// TwinCAT 3 PLC project PLC_Skid
// ProgramVersion: 3.1.4026.20
// libraries:
//   Tc2_ControllerToolbox, * (Beckhoff Automation GmbH)
//   Tc2_SerialCom, * (Beckhoff Automation GmbH)
//   Tc2_Standard, * (Beckhoff Automation GmbH)
//   Tc2_System, * (Beckhoff Automation GmbH)
// project tree:
//   / CyclicTaskController.TcTTO, PlcTask.TcTTO, SerialTask.TcTTO
//   DUTs/ EN_AtlasPumpAction.TcDUT, ST_AtlasPumpCmd.TcDUT, ST_AtlasPumpStatus.TcDUT, ST_MassFlowSensor.TcDUT, ST_PressureSensor.TcDUT, ST_Pumps.TcDUT, ST_Valves.TcDUT
//   GVLs/ GVL.TcGVL, GVL_Params.TcGVL, GVL_Serial.TcGVL, IO.TcGVL
//   POUs/General FBs/ FB_MovingAverage.TcPOU, FB_FirstOrderLP.TcPOU, FB_FlowPathCheck.TcPOU, FB_MassFlowMonitor.TcPOU, FB_PressureMonitor.TcPOU, FB_PulseValve.TcPOU, FB_ScaleAnalog.TcPOU, FB_ValvePOS.TcPOU, FB_PumpCTRL.TcPOU, FB_valveCTRL.TcPOU
//   POUs/ MAIN.TcPOU, SerialComm.TcPOU
//   POUs/PID/ PRG_CONTROLLER_CALL.TcPOU, PRG_FB_CTRL_PI.TcPOU
//   POUs/Status FBs/ FB_CheckValveInputs.TcPOU
//   POUs/UnitOp FBs/ FBUO_OPPUMP_AcetonePrime.TcPOU, FBUO_OPFlowFormation.TcPOU, FBUO_OPPump_SyringeSetup.TcPOU, FBUO_OverPressure.TcPOU, FBUO_OverPressure_EX.TcPOU
// real-time tasks:
//   TASK PlcTask: cycle T#10ms, priority 20, ADS port 350
//   TASK CyclicTaskController: cycle T#10ms, priority 1, ADS port 351
//   TASK SerialTask: cycle T#2ms, priority 2, ADS port 352
// I/O:
//   DEVICE Device 1 (EtherCAT), AmsNetId 192.168.43.43.2.1
//     Term 4 (EK1200) [EK1200-5000 EtherCAT Power supply (2A E-Bus)]
//       Term 20 (ELM3104-0020) [ELM3104-0020 4Ch. Ana. Input +/-20mA, 24 bit, high precision, calibrated]
//       Term 22 (EK1122) [EK1122 2 port EtherCAT junction]
//         Term 23 (EK1100) [EK1100 EtherCAT Coupler (2A E-Bus)]
//           Term 24 (EL1409) [EL1409 16Ch. Dig. Input 24V, 3ms]
//           Term 25 (EL2409) [EL2409 16Ch. Dig. Output 24V, 0.5A]
//           Term 26 (EL3078) [EL3078 8Ch. Ana. Input +/-10V, +/-20mA]
//           Term 27 (EL4078) [EL4078 8Ch. Ana. Output, +/-10V, +/-20mA, 16 Bit]
//           Term 12 (EL9011) [EL9011 End Terminal]
//   DEVICE Device 2 (EtherCAT), AmsNetId 192.168.43.43.3.1
//     Term 4 (IOLITE GATE LATCH v2.00 Bus2) [IOLITE GATE LATCH v2.00 Bus2]
//       Term 5 (IOLITEr 6xSTG Bus2) [IOLITEr 6xSTG Bus2]
//       Term 6 (IOLITEr 6xSTG Bus2) [IOLITEr 6xSTG Bus2]
//       Term 7 (IOLITEr 4xCNT Bus2) [IOLITEr 4xCNT Bus2]
//       Term 8 (IOLITEir 8xRTD-HS Bus2) [IOLITEir 8xRTD-HS Bus2]
//       Term 9 (IOLITEr 32xDI Bus2) [IOLITEr 32xDI Bus2]
//       Term 10 (IOLITEr 16xLV Bus2) [IOLITEr 16xLV Bus2]
//       Term 11 (IOLITEr 16xAO Bus2) [IOLITEr 16xAO Bus2]
//       Term 12 (IOLITEr 32xDO Bus2) [IOLITEr 32xDO Bus2]
//       Term 14 (EL9011) [EL9011 End Terminal]
//     Term 13 (IOLITE GATE LATCH v2.00 Bus2) [IOLITE GATE LATCH v2.00 Bus2]
//       Term 14 (IOLITEr 32xDI Bus2) [IOLITEr 32xDI Bus2]
//       Term 15 (IOLITEr 16xLV Bus2) [IOLITEr 16xLV Bus2]
//       Term 16 (IOLITEr 16xAO Bus2) [IOLITEr 16xAO Bus2]
//       Term 15 (EL9011) [EL9011 End Terminal]
// variable links:
//   (this object) <-> Device 1 (EtherCAT)/Term 4 (EK1200)/Term 20 (ELM3104-0020)
//     PlcTask Inputs/IO.AI_wfiFlowMeter <-> PAI Samples 1 Channel 1/Samples[0]
//   (this object) <-> Device 1 (EtherCAT)/Term 4 (EK1200)/Term 22 (EK1122)/Term 23 (EK1100)/Term 24 (EL1409)
//     PlcTask Inputs/IO.DI1_TestManifold <-> DIP Inputs/Input Channel 1
//     PlcTask Inputs/IO.DI2_TestManifold <-> DIP Inputs/Input Channel 2
//   (this object) <-> Device 1 (EtherCAT)/Term 4 (EK1200)/Term 22 (EK1122)/Term 23 (EK1100)/Term 26 (EL3078)
//     PlcTask Inputs/IO.AI1_TestManifold <-> AI Standard (Real32) Channel 1/Value (Real32)
//   (this object) <-> Device 1 (EtherCAT)/Term 4 (EK1200)/Term 22 (EK1122)/Term 23 (EK1100)/Term 27 (EL4078)
//     PlcTask Outputs/IO.AO1_TestManifold <-> AO Standard (Real32) Channel 1/Value (Real32)
//   (this object) <-> Device 2 (EtherCAT)/Term 13 (IOLITE GATE LATCH v2.00 Bus2)/Term 14 (IOLITEr 32xDI Bus2)
//     PlcTask Inputs/IO.DI1_FormManifold <-> AI TxPDO-Map/DI21
//     PlcTask Inputs/IO.DI2_FormManifold <-> AI TxPDO-Map/DI22
//     PlcTask Inputs/IO.DI1_SuspManifold <-> AI TxPDO-Map/DI17
//     PlcTask Inputs/IO.DI2_SuspManifold <-> AI TxPDO-Map/DI18
//     PlcTask Inputs/IO.DI1_dilutionDiV <-> AI TxPDO-Map/DI13
//     PlcTask Inputs/IO.DI2_dilutionDiV <-> AI TxPDO-Map/DI14
//     PlcTask Inputs/IO.DI1_dilutionSV <-> AI TxPDO-Map/DI1
//     PlcTask Inputs/IO.DI2_dilutionSV <-> AI TxPDO-Map/DI2
//     PlcTask Inputs/IO.DI1_formDrain <-> AI TxPDO-Map/DI9
//     PlcTask Inputs/IO.DI2_formDrain <-> AI TxPDO-Map/DI10
//     PlcTask Inputs/IO.DI1_wfiBypassIn <-> AI TxPDO-Map/DI11
//     PlcTask Inputs/IO.DI2_wfiBypassIn <-> AI TxPDO-Map/DI12
//     PlcTask Inputs/IO.DI1_wfiBypassOut <-> AI TxPDO-Map/DI19
//     PlcTask Inputs/IO.DI2_wfiBypassOut <-> AI TxPDO-Map/DI20
//     PlcTask Inputs/IO.DI1_wfiFilterIn <-> AI TxPDO-Map/DI15
//     PlcTask Inputs/IO.DI2_wfiFilterIn <-> AI TxPDO-Map/DI16
//     PlcTask Inputs/IO.DI1_wfiFilterOut <-> AI TxPDO-Map/DI23
//     PlcTask Inputs/IO.DI2_wfiFilterOut <-> AI TxPDO-Map/DI24
//     PlcTask Inputs/IO.DI1_wfiSV <-> AI TxPDO-Map/DI3
//     PlcTask Inputs/IO.DI2_wfiSV <-> AI TxPDO-Map/DI4
//   (this object) <-> Device 2 (EtherCAT)/Term 13 (IOLITE GATE LATCH v2.00 Bus2)/Term 15 (IOLITEr 16xLV Bus2)
//     PlcTask Inputs/IO.AI1_FormManifold <-> UnBuf TxPDO-Map/u9
//     PlcTask Inputs/IO.AI1_SuspManifold <-> UnBuf TxPDO-Map/u11
//     PlcTask Inputs/IO.AI1_dilutionDiV <-> UnBuf TxPDO-Map/u12
//     PlcTask Inputs/IO.AI1_dilutionSV <-> UnBuf TxPDO-Map/u1
//     PlcTask Inputs/IO.AI1_formDrain <-> UnBuf TxPDO-Map/u8
//     PlcTask Inputs/IO.AI1_wfiBypassIn <-> UnBuf TxPDO-Map/u7
//     PlcTask Inputs/IO.AI1_wfiBypassOut <-> UnBuf TxPDO-Map/u10
//     PlcTask Inputs/IO.AI1_wfiFilterIn <-> UnBuf TxPDO-Map/u5
//     PlcTask Inputs/IO.AI1_wfiFilterOut <-> UnBuf TxPDO-Map/u6
//     PlcTask Inputs/IO.AI1_wfiSV <-> UnBuf TxPDO-Map/u2
//   (this object) <-> Device 2 (EtherCAT)/Term 13 (IOLITE GATE LATCH v2.00 Bus2)/Term 16 (IOLITEr 16xAO Bus2)
//     CyclicTaskController Outputs/IO.AO_wfiPump <-> AO RxPDO-Map/AO 3
//     PlcTask Outputs/IO.AO1_FormManifold <-> AO RxPDO-Map/AO 9
//     PlcTask Outputs/IO.AO1_SuspManifold <-> AO RxPDO-Map/AO 11
//     PlcTask Outputs/IO.AO1_dilutionDiV <-> AO RxPDO-Map/AO 12
//     PlcTask Outputs/IO.AO1_dilutionSV <-> AO RxPDO-Map/AO 1
//     PlcTask Outputs/IO.AO1_formDrain <-> AO RxPDO-Map/AO 8
//     PlcTask Outputs/IO.AO1_wfiBypassIn <-> AO RxPDO-Map/AO 7
//     PlcTask Outputs/IO.AO1_wfiBypassOut <-> AO RxPDO-Map/AO 10
//     PlcTask Outputs/IO.AO1_wfiFilterIn <-> AO RxPDO-Map/AO 5
//     PlcTask Outputs/IO.AO1_wfiFilterOut <-> AO RxPDO-Map/AO 6
//     PlcTask Outputs/IO.AO1_wfiSV <-> AO RxPDO-Map/AO 2
//   (this object) <-> Device 2 (EtherCAT)/Term 4 (IOLITE GATE LATCH v2.00 Bus2)/Term 12 (IOLITEr 32xDO Bus2)
//     CyclicTaskController Outputs/IO.DO_wfiPump <-> DO RxPDO-Map/LED 3
//   (this object) <-> Device 2 (EtherCAT)/Term 4 (IOLITE GATE LATCH v2.00 Bus2)/Term 6 (IOLITEr 6xSTG Bus2)
//     PlcTask Inputs/IO.AI_wfiPressureSensor <-> UnBuf TxPDO-Map/u1

CONFIGURATION PLC_Skid
    RESOURCE PLC ON TwinCAT3
        TASK CyclicTaskController(INTERVAL := T#10ms, PRIORITY := 1);
        TASK PlcTask(INTERVAL := T#10ms, PRIORITY := 20);
        TASK SerialTask(INTERVAL := T#2ms, PRIORITY := 2);
        PROGRAM PRG_CONTROLLER_CALL WITH CyclicTaskController : PRG_CONTROLLER_CALL;
        PROGRAM MAIN WITH PlcTask : MAIN;
        PROGRAM SerialComm WITH SerialTask : SerialComm;
    END_RESOURCE
END_CONFIGURATION

// ---- DUTs/EN_AtlasPumpAction.TcDUT
{attribute 'qualified_only'}
{attribute 'strict'}
{attribute 'to_string'}
TYPE EN_AtlasPumpAction :
(
    IDLE := 0,
    STOP_LEFT,
	STOP_RIGHT,
    PAUSE_LEFT,
    PAUSE_RIGHT,
	UNPAUSE_LEFT,
	UNPAUSE_RIGHT,
    EMPTY_LEFT_FAST,
    EMPTY_RIGHT_FAST,
    FILL_LEFT_FAST,
    FILL_RIGHT_FAST,
	EMPTY_LEFT_PRIME,
    EMPTY_RIGHT_PRIME,
    FILL_LEFT_PRIME,
    FILL_RIGHT_PRIME,
	CONTINUOUS
);
END_TYPE

// ---- DUTs/ST_AtlasPumpCmd.TcDUT
TYPE ST_AtlasPumpCmd :
STRUCT
(* Basic Controls *)
    StopLeft        : STRING := 'X0';
	StopRight        : STRING := 'X1';
    PauseLeft       : STRING := 'W0';
	PauseRight       : STRING := 'W1';
    UnpauseLeft     : STRING := 'U0';
	UnpauseRight     : STRING := 'U1';
    (* 15ml/min Port 2 Commands *)
    (* Format: [Command][Volume/Rate] [Port] *)
    EmptyLeft_FAST   	: STRING := 'E0 70000 2';
    EmptyRight_FAST  	: STRING := 'E1 70000 2';
    FillLeft_FAST    	: STRING := 'F0 70000 1';
    FillRight_FAST		: STRING := 'F1 70000 1';
	EmptyLeft_PRIME   	: STRING := 'E0 40000 2';
    EmptyRight_PRIME  	: STRING := 'E1 40000 2';
    FillLeft_PRIME    	: STRING := 'F0 40000 1';
    FillRight_PRIME   	: STRING := 'F1 40000 1';
	CONTINUOUS		  	: STRING := 'C 35000 2 1 0 0';
END_STRUCT
END_TYPE

// ---- DUTs/ST_AtlasPumpStatus.TcDUT
TYPE ST_AtlasPumpStatus :
STRUCT
    (* Parsed from Status Response: #Sn <error> <state> <vol_remain> <movements> <cumul_vol> <flow_rate> <node1> <node2> <total_cumul> *)

    ErrorCode        : INT;         // 0=OK, 1=busy, 2=invalid pump, 3=failure, 4=invalid port, 5=invalid command
    CurrentState     : INT;         // 1=PUMPS_BUSY, 6=PUMPS_IDLE
    VolumeRemaining  : LREAL;       // ul - raw volume remaining from pump (has offset)
    VolumeRemainingCorrected : LREAL; // ul - corrected volume remaining (0 = empty, SyringeSize = full)
    SyringeMovements : DINT;        // Number of syringe movements
    CumulativeVolume : LREAL;       // ul - cumulative volume pumped (may reset)
    CurrentFlowRate  : LREAL;       // ul/min
    NodeSensor1      : STRING(20);  // Node sensor value 1 (or '?' if no node)
    NodeSensor2      : STRING(20);  // Node sensor value 2 (or '?' if no node)
    TotalCumulativeVol : LREAL;     // ul - total cumulative volume (firmware 1.4.26+, persists)

    (* Status Flags *)
    Valid            : BOOL;        // TRUE if last parse succeeded
    IsBusy           : BOOL;        // TRUE if CurrentState = 1 (PUMPS_BUSY)
    IsIdle           : BOOL;        // TRUE if CurrentState = 6 (PUMPS_IDLE)
    HasError         : BOOL;        // TRUE if ErrorCode <> 0

END_STRUCT
END_TYPE

// ---- DUTs/ST_MassFlowSensor.TcDUT
TYPE ST_MassFlowSensor :
STRUCT
	Name : STRING[20];			// Sensor name
	ID : INT;					// Sensor index
	RawValue : REAL;			// Raw input converted from DINT to REAL
	ScaledValue : REAL;			// Scaled engineering units (computed by FB)
	InputMin : REAL;			// Raw input minimum (e.g., 0.0)
	InputMax : REAL;			// Raw input maximum (e.g., 8388607.0 for 24-bit)
	OutputMin : REAL;			// Scaled output minimum (e.g., 0.0)
	OutputMax : REAL;			// Scaled output maximum (e.g., 4500.0 g/min)
	RangeError : BOOL;			// TRUE if raw input outside expected range
	Status : INT;				// 0=OK, 1=Fault
END_STRUCT
END_TYPE

// ---- DUTs/ST_PressureSensor.TcDUT
TYPE ST_PressureSensor :
STRUCT
	Name : STRING[20];			// Sensor name
	ID : INT;					// Sensor index
	RawValue : REAL;			// Raw 4-20mA input from IO
	ScaledValue : REAL;			// Scaled engineering units, unfiltered (computed by FB)
	FilteredValue : REAL;		// Filtered scaled value (used for control/protection)
	FilterTimeConst : REAL;		// Low-pass filter time constant in seconds (0.0 = no filtering)
	InputMin : REAL;			// Raw input minimum (e.g., 4.0)
	InputMax : REAL;			// Raw input maximum (e.g., 20.0)
	OutputMin : REAL;			// Scaled output minimum (e.g., 0.0)
	OutputMax : REAL;			// Scaled output maximum (e.g., 30.0)
	RangeError : BOOL;			// TRUE if raw input outside expected range
	Status : INT;				// 0=OK, 1=Fault
END_STRUCT
END_TYPE

// ---- DUTs/ST_Pumps.TcDUT
TYPE ST_Pumps :
STRUCT
	Name : STRING[20]; 		// Pump Name
	ID : INT;					// Pump index
	IsOn : BOOL;				// Command: TRUE = pump active
	CMDVoltage : REAL;			// Command: speed setpoint 0-10V
	ControllerIsOn : BOOL;			// Allows for PID Control
	ControllerSetppoint : REAL;		//Setpoint mass flow rate in g/min
	DO1 : BOOL := FALSE;				// Output: digital on/off (computed by FB_PumpCTRL)
	AO1 : REAL := 0;				// Output: analog voltage (computed by FB_PumpCTRL)
	PressureValue : REAL;			// Current pressure reading (mapped from sensor in MAIN)
	PressureLimit : REAL;			// Overpressure trip threshold (0.0 = no check)
	OverPressure : BOOL;			// Latching overpressure flag (clear from HMI to reset)
	FlowPathOpen : BOOL;			// TRUE if required flow path valves are confirmed open
	Status : INT;				// 0=OK, 1=Fault
END_STRUCT
END_TYPE

// ---- DUTs/ST_Valves.TcDUT
TYPE ST_Valves :
STRUCT
    Name : WSTRING(80); // Descriptive name (e.g., 'ValveA', 'InletValve1')
	ID : INT;	// Valve Index
    DI1 : BOOL; // Valve open feedback (if True Valve Open)
    DI2 : BOOL; // Valve closed feedback (if True Valve Close)
    DO1 : BOOL; // Valve Initialization Signal
    AI1 : REAL; // Valve position (0-10V)
    AO1 : REAL; // Valve setpoint (0-10V)
    State : INT; // Operating state (0=Off, 1=Open/Close, 2=OpenLoop, 3=PID)
    isOpen : BOOL; // HMI open/close input
    Setpoint : REAL; // Setpoint for OpenLoop or PID (0-10V)
    PV : REAL; // Process Variable for PID
    Output : REAL; // PID output (0-10V)
	Status : INT; // Diagnostic status (0 = OK, 1 = Fault)
END_STRUCT
END_TYPE

// ---- GVLs/GVL.TcGVL
VAR_GLOBAL CONSTANT
	valveCount : INT := 11;
	sValveNames : ARRAY[1..valveCount] OF WSTRING := 	["Dilution Selector", 
														"WFI Selector", 
														"Formation Drain", 
														"WFI Filter Bypass Inlet",
														"WFI Filter Inlet",
														"WFI Filter Outlet",
														"WFI Filter Bypass Outlet",
														"Dilution Diverter",
														"Formation Manifold",
														"Suspension Manifold",
														"Test Manifold"];													
stValveID : ARRAY[1..valveCount] OF INT := 	[1, 	// Dilution Selector
											 2, 		// WFI Selector,
											 3, 		// Formation Drain,
											 4, 		// WFI Filter Bypass Inlet,
											 5, 		// WFI Filter Inlet,
											 6, 		// WFI Filter Outlet,
											 7, 		// WFI Filter Bypass Outlet,
											 8, 		// Dilution Diverter,
											 9, 		// Formation Manifold,
											 10, 	// Suspension Manifold,
											 11		// Test Manifold
											];
											
pumpCount : INT := 2;
sPumpNames : ARRAY[1..pumpCount] OF WSTRING := 		
	["WFI Pump", "Suspension Pump"];

pressureSensorCount : INT := 3;
sPressureSensorNames : ARRAY[1..pressureSensorCount] OF WSTRING :=
	["WFI Pressure", "Suspension Pressure", "TFF Outlet Pressure"];

massFlowSensorCount : INT := 3;
sMassFlowSensorNames : ARRAY[1..massFlowSensorCount] OF WSTRING :=
	["WFI Mass Flow", "Suspension Mass Flow", "Discharge Flow"];
	
	
END_VAR

VAR_GLOBAL

	myText 		: STRING(16) := 'Type';
	myNum		: REAL := 0;
	avg10WFI_MassFlowRate : REAL;
	
	fSetpointValueToScope			: LREAL;
	fActualValueToScope				: LREAL;
	fOutToScope						: LREAL;
	
END_VAR

// ---- GVLs/GVL_Params.TcGVL
{attribute 'qualified_only'}
VAR_GLOBAL
	


END_VAR

// ---- GVLs/GVL_Serial.TcGVL
{attribute 'qualified_only'}
VAR_GLOBAL
    (* I/O variables for a PC-COM port *)
    stIn_PcCom      AT %I*  : PcComInData;  (* linked to the port in the TwinCAT System Manager *)
    stOut_PcCom     AT %Q*  : PcComOutData; (* linked to the port in the TwinCAT System Manager *)
    RxBufferPcCom           : ComBuffer;    (* Receive data buffer *)
    TxBufferPcCom           : ComBuffer;    (* Transmit data buffer *)

    (* PC Control *)
    bEnablePCControl    : BOOL := FALSE;    // Set TRUE to enable PC Control mode
    sCommandString      : STRING := '';     // Manual command string (set before bStartCommand)
    bStartCommand       : BOOL;             // Trigger to send manual command via sCommandString
    eSelectedAction     : EN_AtlasPumpAction := EN_AtlasPumpAction.IDLE;

    (* Pump Status - Updated every 50ms per axis (100ms total cycle) *)
    stPumpStatus        : ARRAY[0..1] OF ST_AtlasPumpStatus;  // Status for axis 0 and axis 1
    bStatusPollingActive: BOOL := FALSE;    // TRUE when status polling is running

    (* Syringe Configuration - used to correct VolumeRemaining offset *)
    (* Each axis may have a different "full" reference point from the pump *)
    (* Axis 0: Full=5000, Empty=-20000  -> Offset = 20000 (or SyringeSize - FullRef) *)
    (* Axis 1: Full=10000, Empty=-15000 -> Offset = 15000 (or SyringeSize - FullRef) *)
    (* Corrected = Raw + Offset, so that Full=SyringeSize, Empty=0 *)
    rSyringeSize        : ARRAY[0..1] OF LREAL := [25000.0, 25000.0];  // ul - syringe size for each axis
    rFullReference      : ARRAY[0..1] OF LREAL := [5000.0, 10000.0];   // ul - raw value when syringe is full

END_VAR

// ---- GVLs/IO.TcGVL
{attribute 'qualified_only'}
VAR_GLOBAL
	

//----------------------------------DO Place Holder INIT valve 1 -------------------------------------------------//
	//AO1 AT %Q* : REAL;
	DO1 AT %Q* : BOOL;
//---------------------------------------------------------------------------------------------------------------//
	
//---------------------------------- PUMP MAPPING -------------------------------------------------//
	// WFI Pump (index 1)
	DO_wfiPump AT %Q* : BOOL;			// Digital Output for turning pump on and off
	AO_wfiPump AT %Q* : REAL;			// Analog Output for pump speed control
	// Suspension Pump (index 2) - not yet connected
	// DO_suspPump AT %Q* : BOOL;		// Digital Output for turning pump on and off
	// AO_suspPump AT %Q* : REAL;		// Analog Output for pump speed control
//-------------------------------------------------------------------------------------------------//

//---------------------------------- PRESSURE SENSOR MAPPING ----------------------------------------//
	// WFI Pressure Sensor (index 1)
	AI_wfiPressureSensor AT %I* : REAL;			// Analog Input for WFI pressure sensor (4-20mA)
	// Suspension Pressure Sensor (index 2) - not yet connected
	// AI_suspPressureSensor AT %I* : REAL;
	// TFF Outlet Pressure Sensor (index 3) - not yet connected
	// AI_tffOutletPressureSensor AT %I* : REAL;
//-------------------------------------------------------------------------------------------------//

//---------------------------------- MASS FLOW METER MAPPING ------------------------------------------//
	// WFI Mass Flow Meter (index 1)
	AI_wfiFlowMeter AT %I* : DINT;				// Coriolis meter raw input (24-bit DINT)
	// Suspension Mass Flow Meter (index 2) - not yet connected
	// AI_suspMassFlowMeter AT %I* : DINT;
	// Discharge Flow Meter (index 3) - not yet connected
	// AI_dischargeFlowMeter AT %I* : DINT;
//-------------------------------------------------------------------------------------------------//

//---------------------------------- VALVE MAPPING ------------------------------------------------//
	// IOs Dilution Selector Valve (SV)
    DI1_dilutionSV AT %I* : BOOL; 		// Digital Input 1 Closed Feedback
    DI2_dilutionSV AT %I* : BOOL; 		// Digital Input 2 Open Feedback
    AI1_dilutionSV AT %I* : REAL;  		// Analog Input 1 Valve Position Feedback
    DO1_dilutionSV AT %Q* : BOOL; 		// Digital Output 1 Valve Initialization
    AO1_dilutionSV AT %Q* : REAL; 		// Analog Output 1 Valve Position Control Variable (0-10V)
    
    // IOs WFI Selector Valve (SV) 
    DI1_wfiSV AT %I* : BOOL;      		// Digital Input 1 Closed Feedback
    DI2_wfiSV AT %I* : BOOL;      		// Digital Input 2 Open Feedback
    AI1_wfiSV AT %I* : REAL;       		// Analog Input 1 Valve Position Feedback
    DO1_wfiSV AT %Q* : BOOL;     		// Digital Output 1 Valve Initialization
    AO1_wfiSV AT %Q* : REAL;      		// Analog Output 1 Valve Position Control Variable (0-10V)

	// IOs Formation Drain Valve 
    DI1_formDrain AT %I* : BOOL;      	// Digital Input 1 Closed Feedback
    DI2_formDrain AT %I* : BOOL;      	// Digital Input 2 Open Feedback
    AI1_formDrain AT %I* : REAL;       	// Analog Input 1 Valve Position Feedback
    DO1_formDrain AT %Q* : BOOL;     	// Digital Output 1 Valve Initialization
    AO1_formDrain AT %Q* : REAL;      	// Analog Output 1 Valve Position Control Variable (0-10V)
	
	// IOs WFI Bypass Inlet Valve
    DI1_wfiBypassIn AT %I* : BOOL;      // Digital Input 1 Closed Feedback
    DI2_wfiBypassIn AT %I* : BOOL;      // Digital Input 2 Open Feedback
    AI1_wfiBypassIn AT %I* : REAL;      // Analog Input 1 Valve Position Feedback
    DO1_wfiBypassIn AT %Q* : BOOL;     	// Digital Output 1 Valve Initialization
    AO1_wfiBypassIn AT %Q* : REAL;      // Analog Output 1 Valve Position Control Variable (0-10V)
	
		// IOs WFI Filter Inlet Valve
    DI1_wfiFilterIn AT %I* : BOOL;      // Digital Input 1 Closed Feedback
    DI2_wfiFilterIn AT %I* : BOOL;      // Digital Input 2 Open Feedback
    AI1_wfiFilterIn AT %I* : REAL;      // Analog Input 1 Valve Position Feedback
    DO1_wfiFilterIn AT %Q* : BOOL;     	// Digital Output 1 Valve Initialization
    AO1_wfiFilterIn AT %Q* : REAL;      // Analog Output 1 Valve Position Control Variable (0-10V)
	
		// IOs WFI Filter Outlet Valve
    DI1_wfiFilterOut AT %I* : BOOL;      // Digital Input 1 Closed Feedback
    DI2_wfiFilterOut AT %I* : BOOL;      // Digital Input 2 Open Feedback
    AI1_wfiFilterOut AT %I* : REAL;      // Analog Input 1 Valve Position Feedback
    DO1_wfiFilterOut AT %Q* : BOOL;     	// Digital Output 1 Valve Initialization
    AO1_wfiFilterOut AT %Q* : REAL;      // Analog Output 1 Valve Position Control Variable (0-10V)
	
		// IOs WFI Bypass Outlet Valve
    DI1_wfiBypassOut AT %I* : BOOL;      // Digital Input 1 Closed Feedback
    DI2_wfiBypassOut AT %I* : BOOL;      // Digital Input 2 Open Feedback
    AI1_wfiBypassOut AT %I* : REAL;      // Analog Input 1 Valve Position Feedback
    DO1_wfiBypassOut AT %Q* : BOOL;     	// Digital Output 1 Valve Initialization
    AO1_wfiBypassOut AT %Q* : REAL;      // Analog Output 1 Valve Position Control Variable (0-10V)
	
		// IOs Dilution Diverter Valve
    DI1_dilutionDiV AT %I* : BOOL;      // Digital Input 1 Closed Feedback
    DI2_dilutionDiV AT %I* : BOOL;      // Digital Input 2 Open Feedback
    AI1_dilutionDiV AT %I* : REAL;      // Analog Input 1 Valve Position Feedback
    DO1_dilutionDiV AT %Q* : BOOL;     	// Digital Output 1 Valve Initialization
    AO1_dilutionDiV AT %Q* : REAL;      // Analog Output 1 Valve Position Control Variable (0-10V)
	
		// IOs Formation Manifold Valve
    DI1_FormManifold AT %I* : BOOL;      // Digital Input 1 Closed Feedback
    DI2_FormManifold AT %I* : BOOL;      // Digital Input 2 Open Feedback
    AI1_FormManifold AT %I* : REAL;      // Analog Input 1 Valve Position Feedback
    DO1_FormManifold AT %Q* : BOOL;     	// Digital Output 1 Valve Initialization
    AO1_FormManifold AT %Q* : REAL;      // Analog Output 1 Valve Position Control Variable (0-10V)
	
		// IOs Suspension Manifold Valve
    DI1_SuspManifold AT %I* : BOOL;      // Digital Input 1 Closed Feedback
    DI2_SuspManifold AT %I* : BOOL;      // Digital Input 2 Open Feedback
    AI1_SuspManifold AT %I* : REAL;      // Analog Input 1 Valve Position Feedback
    DO1_SuspManifold AT %Q* : BOOL;     	// Digital Output 1 Valve Initialization
    AO1_SuspManifold AT %Q* : REAL;      // Analog Output 1 Valve Position Control Variable (0-10V)
	
			// IOs Test Manifold Valve
    DI1_TestManifold AT %I* : BOOL;      // Digital Input 1 Closed Feedback
    DI2_TestManifold AT %I* : BOOL;      // Digital Input 2 Open Feedback
    AI1_TestManifold AT %I* : REAL;      // Analog Input 1 Valve Position Feedback (4-20ma)
    DO1_TestManifold AT %Q* : BOOL;     	// Digital Output 1 Valve Initialization
    AO1_TestManifold AT %Q* : REAL;      // Analog Output 1 Valve Position Control Variable (4-20ma)
//-------------------------------------------------------------------------------------------------//

END_VAR

// ---- POUs/PID/PRG_CONTROLLER_CALL.TcPOU
PROGRAM PRG_CONTROLLER_CALL

VAR
	
	stPumps 	: ARRAY[1..GVL.pumpCount] OF ST_Pumps;
	
	
END_VAR




IF stPumps[1].ControllerIsOn AND stPumps[1].IsOn THEN
	IO.DO_wfiPump 					:= TRUE;
	PRG_FB_CTRL_PI();

	ELSE
	IO.DO_wfiPump := FALSE;
	IO.AO_wfiPump := stPumps[1].ControllerSetppoint := 0;
END_IF

END_PROGRAM

// ---- POUs/PID/PRG_FB_CTRL_PI.TcPOU
PROGRAM PRG_FB_CTRL_PI


VAR
	stPumps 	: ARRAY[1..GVL.pumpCount] OF ST_Pumps;	

	fSetpointValue				: LREAL;
	fActualValue				: LREAL;
	fManSyncValue				: LREAL;
	bSync						: BOOL;

	fOut						: LREAL;
	bHold						: BOOL;

	eMode						: E_CTRL_MODE;
	stCTRL_PI_PARAMS			: ST_CTRL_PI_PARAMS;

	eErrorId					: E_CTRL_ERRORCODES;
	bError						: BOOL;
	bARWactive					: BOOL;

	(* controller  *)
	fbCTRL_PI					: FB_CTRL_PI;

	bInit						: BOOL := TRUE;
	fbTON						: TON;
END_VAR

IF bInit THEN
	(* init parameter struct *)
	stCTRL_PI_PARAMS.tCtrlCycleTime		:= T#10MS;
	stCTRL_PI_PARAMS.tTaskCycleTime		:= T#10MS;
	stCTRL_PI_PARAMS.tTn				:= T#2S;	(* derivative gain Tv				*)
	stCTRL_PI_PARAMS.fKp				:= 2;		(* proportional gain Kp				*)
	stCTRL_PI_PARAMS.fOutMaxLimit		:= 3;  		(* maximum output limit				*)
	stCTRL_PI_PARAMS.fOutMinLimit		:= 0;		(* minimum output limit				*)

	(* set the mode to ACTIVE --> normal operation *)
	eMode := eCTRL_MODE_ACTIVE;

	(* reset the init flag *)
	bInit := FALSE;
END_IF

fSetpointValue := stPumps[1].ControllerSetppoint;
fActualValue := GVL.avg10WFI_MassFlowRate;

(* copy var to scope var *)
fSetpointValueToScope 		:= fSetpointValue;
fActualValueToScope 		:= fActualValue;

(* call controller *)
fbCTRL_PI(		fSetpointValue		:= fSetpointValue,
					fActualValue		:= fActualValue,
					fManSyncValue	:= fManSyncValue,
					bSync				:= bSync,
					eMode				:= eMode,
					bHold				:= bHold,
					stParams			:= stCTRL_PI_PARAMS,
					fOut				=> fOut,
					bARWactive		=> bARWactive,
					eErrorId			=> eErrorId,
					bError				=> bError
				);


(* copy var to scope var *)
fOut := stPumps[1].CMDVoltage;
fOutToScope := fOut;

END_PROGRAM

// ---- POUs/MAIN.TcPOU
PROGRAM MAIN
VAR
//-------------------- Program Initialization Variables ----------------------------//
	i : INT; //Initialization Counter
	CycleCount : INT := 0; // Cycle counter
	Initialized : BOOL := FALSE; // Flag for initialization
	CtrlStatus : INT; // Status output
//----------------------------------------------------------------------------------//


//--------------------------------- Struct Init ------------------------------------//
// Constant array of valve names
	stValves : ARRAY[1..GVL.valveCount] OF ST_Valves;
	stPumps : ARRAY[1..GVL.pumpCount] OF ST_Pumps;
	stPressureSensors : ARRAY[1..GVL.pressureSensorCount] OF ST_PressureSensor;
	stMassFlowSensors : ARRAY[1..GVL.massFlowSensorCount] OF ST_MassFlowSensor;
//----------------------------------------------------------------------------------//


//----------------------------INIT Function Blocks----------------------------------//
	systemCheck_Valves : FB_CheckValveInputs;
	valveCtrl : FB_valveCTRL;
	pumpCtrl : FB_PumpCTRL;
	varPulse : FB_PulseValve;   // Instance of the function block
	unitOp_OverPressure : FBUO_OverPressure;
	unitOp_OverPressureEX : FBUO_OverPressure_EX;
	pressureMonitor : FB_PressureMonitor;
	massFlowMonitor : FB_MassFlowMonitor;
	flowPathCheck_WFI : FB_FlowPathCheck;
	wfi_MassFlowAvg10 : FB_MovingAverage;
	wfi_MassFlowAvg30 : FB_MovingAverage;
	wfi_MassFlowAvg100 : FB_MovingAverage;
//----------------------------------------------------------------------------------//	
	
//---------------------------- General Variables -----------------------------------//
	outputDO1 : BOOL;           // Local output variable
    tPulseTime : TIME := T#1000MS; // Pulse duration
	//avg10WFI_MassFlowRate : REAL;
	avg30WFI_MassFlowRate : REAL;
	avg100WFI_MassFlowRate : REAL;
	
//---------------------INIT Control Variables---------------------------------------//
	hOP_ProcessState			: BOOL	:= TRUE;	// Overpressure process step active
	hOP_ValvesPositionSet	 	: BOOL 	:= TRUE;	// Position Valves
	hOP_PumpActive				: BOOL	:= FALSE;	// Turn on Pump
	hOP_PumpSpeed				: REAL 	:= 0;		// Pump Speed
//----------------------------------------------------------------------------------//

//---------------------INIT Control Variables---------------------------------------//
	hOPEX_ProcessState			: BOOL	:= FALSE;	// Overpressure process step active
	hOPEX_ValvesPositionSet	 	: BOOL 	:= FALSE;	// Position Valves
	hOPEX_PumpActive			: BOOL	:= FALSE;	// Turn on Pump
//----------------------------------------------------------------------------------//

//---------------------Flow Path Definitions---------------------------------------//
	wfiFlowPath_OP		: ARRAY[1..GVL.valveCount] OF INT := [2,5,0,0,0,0,0,0,0,0];
	wfiFlowPath_OPEX	: ARRAY[1..GVL.valveCount] OF INT := [2,4,7,8,9,10,0,0,0,0];
	wfiActiveFlowPath	: ARRAY[1..GVL.valveCount] OF INT;
//----------------------------------------------------------------------------------//


//----------------------------INIT Function Blocks----------------------------------//
	fbSyringeSetup : FBUO_OPPump_SyringeSetup;
	fbAcetonePrime : FBUO_OPPump_AcetonePrime;
	fbFlowFormation : FBUO_OPFlowFormation;
//----------------------------------------------------------------------------------//

///---------------------Organic Phase Setup ---------------------------------------//
OPActive					: BOOL	:= FALSE;
bStartSyringeSetup			: BOOL	:= FALSE;	// Start Syringe Setup Routine
bStartActenePriming			: BOOL	:= FALSE;	// Start Acetone Priming Routine
bStartFlowFormation			: BOOL	:= FALSE;	// Start/Stop Continuous Flow Formation
nAcetoneCycles				: INT	:= 2;
nAcetoneCycle				: INT;	
//----------------------------------------------------------------------------------//

// -----------------------MATLAB Variables for testing ----------------------------//
mtbIN		: INT		:= 1000;
mtbOUT		: INT;
mtbActive	: BOOL		:= FALSE;	
currentValue : REAL := 0;
END_VAR

//------------------------------------Process Code ----------------------------------------//
//---------------------------------- Initialization----------------------------------------//
IF NOT Initialized THEN
    FOR i := 1 TO gvl.valveCount DO
        stValves[i].Name := GVL.sValveNames[i]; // Assign valve names
		stValves[i].ID := GVL.stValveID[i];
        stValves[i].State := 0; // Initialize to Closed
        stValves[i].AO1 := 0.0; // Closed position
        stValves[i].Status := 0; // No faults
        stValves[i].isOpen := FALSE; // Initialize to closed
    END_FOR
	FOR i := 1 TO GVL.pumpCount DO
		stPumps[i].Name := WSTRING_TO_STRING(GVL.sPumpNames[i]);
		stPumps[i].ID := i;
		stPumps[i].IsOn := FALSE;
		stPumps[i].CMDVoltage := 0.0;
		stPumps[i].ControllerIsOn := FALSE;
		stPumps[i].DO1 := FALSE;
		stPumps[i].AO1 := 0.0;
		stPumps[i].PressureValue := 0.0;
		stPumps[i].PressureLimit := 10.0;
		stPumps[i].OverPressure := FALSE;
		stPumps[i].FlowPathOpen := FALSE;
		stPumps[i].Status := 0;
	END_FOR
	FOR i := 1 TO GVL.pressureSensorCount DO
		stPressureSensors[i].Name := WSTRING_TO_STRING(GVL.sPressureSensorNames[i]);
		stPressureSensors[i].ID := i;
		stPressureSensors[i].RawValue := 0.0;
		stPressureSensors[i].ScaledValue := 0.0;
		stPressureSensors[i].FilteredValue := 0.0;
		stPressureSensors[i].FilterTimeConst := 0.1;
		stPressureSensors[i].InputMin := 4.0;
		stPressureSensors[i].InputMax := 20.0;
		stPressureSensors[i].OutputMin := 0.0;
		stPressureSensors[i].OutputMax := 30.0;
		stPressureSensors[i].RangeError := FALSE;
		stPressureSensors[i].Status := 0;
	END_FOR
	FOR i := 1 TO GVL.massFlowSensorCount DO
		stMassFlowSensors[i].Name := WSTRING_TO_STRING(GVL.sMassFlowSensorNames[i]);
		stMassFlowSensors[i].ID := i;
		stMassFlowSensors[i].RawValue := 0.0;
		stMassFlowSensors[i].ScaledValue := 0.0;
		stMassFlowSensors[i].InputMin := 0;
		stMassFlowSensors[i].InputMax := 8388607.0;
		stMassFlowSensors[i].OutputMin := 0.0;
		stMassFlowSensors[i].OutputMax := 4500.0;
		stMassFlowSensors[i].RangeError := FALSE;
		stMassFlowSensors[i].Status := 0;
	END_FOR
    Initialized := TRUE;
END_IF
CycleCount := CycleCount + 1;

//--------------------------------------------------------------------------------------------//


//------------------------------ Valve Position Monitoring -----------------------------------//
systemCheck_Valves(
	fbCheckProcessState := TRUE, 
	fbValves 			:= stValves);
//--------------------------------------------------------------------------------------------//

//------------------------------- Flow Path Check --------------------------------------------//
// Select active flow path based on which operation is running
IF hOP_ProcessState THEN
	wfiActiveFlowPath := wfiFlowPath_OP;
ELSIF hOPEX_ProcessState THEN
	wfiActiveFlowPath := wfiFlowPath_OPEX;
END_IF
// Check if required valves are confirmed open
flowPathCheck_WFI(
	fbRequiredValves := wfiActiveFlowPath,
	fbValves := stValves);
stPumps[1].FlowPathOpen := flowPathCheck_WFI.fbPathOpen;
//------------------------------------------------------------------------------------------//

//------------------------- Overpressure Process (Development Only) --------------------------//
unitOp_OverPressureEX(
	fbOPprocessState 		:= hOPEX_ProcessState,
	fbValvePositionReady 	:= hOPEX_ValvesPositionSet, 
	fbValves 				:= stValves);
//--------------------------------------------------------------------------------------------//


//------------------------- Overpressure Process (Development Only) --------------------------//
unitOp_OverPressure(
	fbOPprocessState 		:= hOP_ProcessState,
	fbValvePositionReady 	:= hOP_ValvesPositionSet, 
	fbValves 				:= stValves,
	fbPumpActive			:=hOP_PumpActive,
	fbPumpSpeed				:= hOP_PumpSpeed);
//--------------------------------------------------------------------------------------------//

//---------------------------------- Atlas Syringe Setup--------------------------------------//
GVL_Serial.bEnablePCControl := OPActive;
IF OPActive THEN
  fbSyringeSetup(
      bEnable := TRUE,
      bStart  := bStartSyringeSetup
  );
//--------------------------------------------------------------------------------------------//  

//---------------------------------- Acetone Priming -----------------------------------------//
  fbAcetonePrime(
      bEnable            := TRUE,
      bStartAcetonePrime := bStartActenePriming,
      nSyringeCycles     := nAcetoneCycles
  );
  // Monitor progress
  nAcetoneCycle := fbAcetonePrime.nCurrentCycle;  // Shows 1, then 2

//---------------------------------- Continuous Flow Formation --------------------------------//
  fbFlowFormation(
      bEnable := TRUE,
      bStart  := bStartFlowFormation
  );
END_IF
//--------------------------------------------------------------------------------------------// 

//OP Routine Status
  IF fbSyringeSetup.bDone THEN
      // Syringes at 12.5ml - ready for operator to attach
  END_IF

  IF fbAcetonePrime.bDone THEN
      // Priming complete, syringes are empty
  END_IF

//------------------------------ Pressure Monitoring ----------------------------------------//
// Pressure Sensor I/O Mapping
stPressureSensors[1].RawValue := IO.AI_wfiPressureSensor;
// stPressureSensors[2].RawValue := IO.AI_suspPressureSensor;       // uncomment when wired
// stPressureSensors[3].RawValue := IO.AI_tffOutletPressureSensor;  // uncomment when wired
pressureMonitor(fbSensors := stPressureSensors);
//---------------------------------------------------------------------------------------------//

//----------------------------- Mass Flow Monitoring -----------------------------------------------------//					
// Mass Flow Sensor I/O Mapping (DINT to REAL conversion at boundary)
stMassFlowSensors[1].RawValue := DINT_TO_REAL(IO.AI_wfiFlowMeter);
// stMassFlowSensors[2].RawValue := DINT_TO_REAL(IO.AI_suspMassFlowMeter);     // uncomment when wired
// stMassFlowSensors[3].RawValue := DINT_TO_REAL(IO.AI_dischargeFlowMeter);    // uncomment when wired
massFlowMonitor(fbSensors := stMassFlowSensors);

// 10-sample moving average for WFI mass flow rate
wfi_MassFlowAvg10(
	fbInputValue := stMassFlowSensors[1].ScaledValue,
	fbSampleSize := 10,
	fbAverageValue => GVL.avg10WFI_MassFlowRate);

// 30-sample moving average for WFI mass flow rate
wfi_MassFlowAvg30(
	fbInputValue := stMassFlowSensors[1].ScaledValue,
	fbSampleSize := 30,
	fbAverageValue => avg30WFI_MassFlowRate);

// 100-sample moving average for WFI mass flow rate
wfi_MassFlowAvg100(
	fbInputValue := stMassFlowSensors[1].ScaledValue,
	fbSampleSize := 100,
	fbAverageValue => avg100WFI_MassFlowRate);
//-----------------------------------------------------------------------------------------------------//

//------------------------------- Pump Control ------------------------------------//
// Map filtered pressure readings to pumps for overpressure protection
stPumps[1].PressureValue := stPressureSensors[1].FilteredValue;	// WFI Pump <- WFI Pressure
stPumps[2].PressureValue := stPressureSensors[2].FilteredValue;	// Suspension Pump <- Suspension Pressure
pumpCtrl(fbPumps := stPumps);
// WFI Pump I/O Mapping (index 1)
IF mtbActive AND NOT stPumps[1].ControllerIsOn THEN
	IO.DO_wfiPump := stPumps[1].DO1;
	IO.AO_wfiPump := stPumps[1].AO1;
	ELSE
	IO.DO_wfiPump := FALSE;
	IO.AO_wfiPump := 0;
END_IF
// Suspension Pump I/O Mapping (index 2) - uncomment when I/O available
// IO.DO_suspPump := stPumps[2].DO1;
// IO.AO_suspPump := stPumps[2].AO1;
//--------------------------------------------------------------------------------------------------------------//

//------------------------------- Matlab Testing ---------------------------------------------------------------//

IF mtbActive AND mtbOut <500 THEN
	mtbOut := mtbOut+mtbIN;
	ELSE
	mtbOut :=0;
END_IF
IO.AO1_TestManifold := currentValue;
//--------------------------------------------------------------------------------------------------------------//

//------------------------------- Valve Init Function (To be refined later) ------------------------------------//
// Correct function block call with inputs
varPulse(Valve := outputDO1, pulseTime := tPulseTime);
// Assign output to global I/O
IO.DO1_dilutionSV := outputDO1;
//-----------------------------------------------------------------------------------------------------//

//-----------------------------Process Code END ----------------------------------------//

END_PROGRAM

// ---- POUs/Status FBs/FB_CheckValveInputs.TcPOU
FUNCTION_BLOCK FB_CheckValveInputs
VAR_INPUT
	fbCheckProcessState :	BOOL;
END_VAR
VAR_IN_OUT
    fbValves : ARRAY[1..GVL.valveCount] OF ST_Valves;
END_VAR
VAR_OUTPUT
	
END_VAR
VAR
	
END_VAR

IF fbCheckProcessState THEN
	fbValves[1].DI1 := IO.DI1_dilutionSV;
	fbValves[1].AI1 := IO.AI1_dilutionSV;
	fbValves[1].DI2 := IO.DI2_dilutionSV;

	fbValves[2].DI1 := IO.DI1_wfiSV;
	fbValves[2].AI1 := IO.AI1_wfiSV;
	fbValves[2].DI2 := IO.DI2_wfiSV;

	fbValves[3].DI1 := IO.DI1_formDrain;
	fbValves[3].AI1 := IO.AI1_formDrain;
	fbValves[3].DI2 := IO.DI2_formDrain;

	fbValves[4].DI1 := IO.DI1_wfiBypassIn;
	fbValves[4].AI1 := IO.AI1_wfiBypassIn;
	fbValves[4].DI2 := IO.DI2_wfiBypassIn;
	
	fbValves[5].DI1 := IO.DI1_wfiFilterIn;
	fbValves[5].AI1 := IO.AI1_wfiFilterIn;
	fbValves[5].DI2 := IO.DI2_wfiFilterIn;
	
	fbValves[6].DI1 := IO.DI1_wfiFilterOut;
	fbValves[6].AI1 := IO.AI1_wfiFilterOut;
	fbValves[6].DI2 := IO.DI2_wfiFilterOut;
	
	fbValves[7].DI1 := IO.DI1_wfiBypassOut;
	fbValves[7].AI1 := IO.AI1_wfiBypassOut;
	fbValves[7].DI2 := IO.DI2_wfiBypassOut;
	
	fbValves[8].DI1 := IO.DI1_dilutionDiV;
	fbValves[8].AI1 := IO.AI1_dilutionDiV;
	fbValves[8].DI2 := IO.DI2_dilutionDiV;
	
	fbValves[9].DI1 := IO.DI1_FormManifold;
	fbValves[9].AI1 := IO.AI1_FormManifold;
	fbValves[9].DI2 := IO.DI2_FormManifold;
	
	fbValves[10].DI1 := IO.DI1_SuspManifold;
	fbValves[10].AI1 := IO.AI1_SuspManifold;
	fbValves[10].DI2 := IO.DI2_SuspManifold;
END_IF

END_FUNCTION_BLOCK

// ---- POUs/General FBs/FB_valveCTRL.TcPOU
FUNCTION_BLOCK FB_valveCTRL
VAR_INPUT
    //fbValveNames : ARRAY[1..GVL.valveCount] OF STRING[20]; // Array of valve names
END_VAR
VAR_IN_OUT
    fbValves : ARRAY[1..GVL.valveCount] OF ST_Valves;   // Array of valve structures
END_VAR
VAR_OUTPUT
    //Status : INT;                             // 0=OK, 1=Valve not found
END_VAR
VAR
    i : INT;                                  // Internal loop variable
END_VAR

// Initialize output
//Status := 0;

// Control valves based on hOpenClose
FOR i := 1 TO gvl.valveCount DO
    //IF fbValves[i].Name = fbValveNames[i] THEN
        CASE fbValves[i].State OF
            1: // Open/Close mode
                IF fbValves[i].isOpen THEN
                    fbValves[i].AO1 := 10.0; // Open
                ELSE
                    fbValves[i].AO1 := 0.0; // Close
                END_IF
            2: // OpenLoop
                fbValves[i].AO1 := fbValves[i].Setpoint;
            3: // PID (Placeholder)
                fbValves[i].AO1 := 0.0;
            ELSE
                fbValves[i].AO1 := 0.0;
                //Status := Status + 2;
        END_CASE
    //ELSE
        //Status := Status + 1;
    //END_IF
END_FOR

END_FUNCTION_BLOCK

// ---- POUs/General FBs/FB_PumpCTRL.TcPOU
FUNCTION_BLOCK FB_PumpCTRL
VAR_INPUT
END_VAR
VAR_IN_OUT
    fbPumps : ARRAY[1..GVL.pumpCount] OF ST_Pumps;   // Array of pump structures
END_VAR
VAR_OUTPUT
END_VAR
VAR
    i : INT;                                  // Internal loop variable
END_VAR

// Pump control - open loop voltage command with overpressure protection
FOR i := 1 TO GVL.pumpCount DO
	// Overpressure latch: trips when pressure >= limit, stays latched until cleared externally
	IF fbPumps[i].PressureLimit > 0.0 AND fbPumps[i].PressureValue >= fbPumps[i].PressureLimit THEN
		fbPumps[i].OverPressure := TRUE;
	END_IF

	// Control pump output (safety checks: overpressure, flow path)
	IF fbPumps[i].OverPressure THEN
		fbPumps[i].DO1 := FALSE;
		fbPumps[i].AO1 := 0.0;
	ELSIF NOT fbPumps[i].FlowPathOpen THEN
		fbPumps[i].DO1 := FALSE;
		fbPumps[i].AO1 := 0.0;
	ELSIF fbPumps[i].IsOn THEN
		fbPumps[i].DO1 := TRUE;
		fbPumps[i].AO1 := LIMIT(0.0, fbPumps[i].CMDVoltage, 10.0);
	ELSE
		fbPumps[i].DO1 := FALSE;
		fbPumps[i].AO1 := 0.0;
	END_IF
END_FOR

END_FUNCTION_BLOCK

// ---- POUs/General FBs/FB_PulseValve.TcPOU
FUNCTION_BLOCK FB_PulseValve
VAR_INPUT
	Valve : REFERENCE TO BOOL;  // Reference to BOOL output (e.g., output1)
    pulseTime : TIME;               // Pulse duration
END_VAR
VAR_OUTPUT
	bDone : BOOL;               // TRUE when pulse completes
    bBusy : BOOL;               // TRUE during pulse
END_VAR
VAR
	timer : TON;
    bTriggerOld : BOOL;
    bRising : BOOL;
END_VAR

// Rising edge detection
bRising := Valve AND NOT bTriggerOld;
bTriggerOld := Valve;

// Start timer on rising edge
IF bRising THEN
    timer(IN := TRUE, PT := pulseTime);
END_IF;

//Execute Timer
timer();

// Output control: Valve ON during timing, OFF after
IF timer.IN AND NOT timer.Q THEN
Valve := timer.IN;
ELSE
VALVE := FALSE;
END_IF

// Reset and signal done
IF timer.Q THEN
    timer.IN := FALSE;
    bDone := TRUE;
END_IF;

bBusy := timer.IN;

END_FUNCTION_BLOCK

// ---- POUs/UnitOp FBs/FBUO_OverPressure.TcPOU
FUNCTION_BLOCK FBUO_OverPressure
VAR_INPUT
    fbOPprocessState 		: BOOL;
    fbValvePositionReady 	: BOOL;
	fbPumpActive 			: BOOL;
	fbPumpSpeed				: REAL;
END_VAR
VAR_IN_OUT
    fbValves : ARRAY[1..GVL.valveCount] OF ST_Valves;
END_VAR
VAR_OUTPUT
	
END_VAR
VAR
    valveIndexOpen : ARRAY[1..GVL.valveCount] OF INT := [2,5];
	numValvesToOpen : INT := 10;
	valveIndexClose : ARRAY[1..GVL.valveCount] OF INT := [2,5];
	numValvesToClose : INT := 10;
    targetState : INT;
    targetOpenClose : BOOL;
	fbValvePos : FB_ValvePOS;
	valveCtrl : FB_valveCTRL;
	valveIndex: INT;
END_VAR

IF fbOPprocessState THEN
	
	fbValvePos(fbValveIndexOpen := valveIndexOpen,
            fbNumValvesToOpen := numValvesToOpen,
			fbValveIndexClose := valveIndexClose,
            fbNumValvesToClose := numValvesToClose,
            fbValves := fbValves,
			fbProcessValves2Open := fbValvePositionReady);
    
    ValveCtrl(fbValves := fbValves);
    IO.AO1_dilutionSV := fbValves[1].AO1;
    IO.AO1_wfiSV := fbValves[2].AO1;
    IO.AO1_formDrain := fbValves[3].AO1;
    IO.AO1_wfiBypassIn := fbValves[4].AO1;
	IO.AO1_wfiFilterIn := fbValves[5].AO1;
	IO.AO1_wfiFilterOut := fbValves[6].AO1;
	IO.AO1_wfiBypassOut := fbValves[7].AO1;
	IO.AO1_dilutionDiV := fbValves[8].AO1;
	IO.AO1_FormManifold := fbValves[9].AO1;
	IO.AO1_SuspManifold := fbValves[10].AO1;
	
	
	
//-----------------------PUMP Control ----------------------//	
// 	IF fbPumpActive THEN
// 	outputAO3 := IO.AO3 := 5;
// 		GVL.DO_wfiPump := fbPumpActive;
// 		GVL.AO_wfiPump := fbPumpSpeed;
// 	ELSE
// 		GVL.DO_wfiPump := fbPumpActive;
// 		GVL.AO_wfiPump := 0;
// 	END_IF	
//---------------------------------------------------------//	
END_IF

END_FUNCTION_BLOCK

// ---- POUs/General FBs/FB_ValvePOS.TcPOU
FUNCTION_BLOCK FB_ValvePOS
VAR_INPUT
    fbValveIndexOpen : ARRAY[1..GVL.valveCount] OF INT;  // Array of valve IDs for opening sequence
    fbNumValvesToOpen : INT;                              // How many valves to open
    fbValveIndexClose : ARRAY[1..GVL.valveCount] OF INT; // Array of valve IDs for closing sequence
    fbNumValvesToClose : INT;                             // How many valves to close
    fbProcessValves2Open : BOOL;                          // TRUE=Open sequence, FALSE=Close sequence
END_VAR

VAR_IN_OUT
    fbValves : ARRAY[1..GVL.valveCount] OF ST_Valves;    // Valve array
END_VAR

VAR_OUTPUT
    fbSequenceComplete : BOOL;                            // TRUE when all valves positioned
    fbSequenceActive : BOOL;                              // TRUE while sequencing in progress
    fbCurrentValveNum : INT;                              // Current valve being positioned (1 to fbNumValvesToPosition)
    fbFaultTimeout : BOOL;                                // TRUE if a valve failed to move
END_VAR

VAR
    // State machine
    sequenceState : INT := 0;                             // 0=Idle, 1=Command, 2=WaitEdge, 3=Delay, 4=Advance
    currentValveIndex : INT := 1;                         // Which valve in sequence array (1 to fbNumValvesToOpen/Close)
    currentValveArrayPos : INT := 0;                      // Position in fbValves array where valve was found
    isOpeningMode : BOOL := FALSE;                        // TRUE=Opening sequence, FALSE=Closing sequence
    lastProcessCommand : BOOL := FALSE;                   // Previous state of fbProcessValves2Open for edge detection

    // Edge detection for DI2 (closed feedback)
    lastDI2State : BOOL := FALSE;                         // Previous scan DI2 value
    valveStartedMoving : BOOL := FALSE;                   // Flag: edge detected

    // Timers
    delayTimer : TON;                                     // 0.5s delay between valve movements
    timeoutTimer : TON;                                   // Timeout if valve doesn't start moving

    // Constants
    VALVE_MOVE_DELAY : TIME := T#750MS;                  // Delay between commanding valves
    VALVE_MOVE_TIMEOUT : TIME := T#5S;                    // Max time to wait for valve to start moving

    // Internal
    i : INT;                                              // Loop counter
    valveFound : BOOL;                                    // Flag for valve lookup
    numValvesInSequence : INT;                            // Total valves in current sequence
END_VAR

// State Machine for Sequential Valve Positioning with Timing Delays
// Supports separate opening and closing sequences with different orders
// Prevents commanding next valve until current valve starts moving + delay

CASE sequenceState OF

    //---------- State 0: Idle/Ready ----------//
    0:
        fbSequenceActive := FALSE;
        fbSequenceComplete := FALSE;
        fbFaultTimeout := FALSE;

        // Reset timers
        delayTimer(IN := FALSE);
        timeoutTimer(IN := FALSE);

        // Detect rising edge on fbProcessValves2Open (start opening sequence)
        IF fbProcessValves2Open AND NOT lastProcessCommand THEN
            // Start opening sequence
            isOpeningMode := TRUE;
            currentValveIndex := 1;
            numValvesInSequence := fbNumValvesToOpen;
            fbSequenceActive := TRUE;
            fbSequenceComplete := FALSE;
            sequenceState := 1;  // Go to command first valve
        END_IF

        // Detect falling edge on fbProcessValves2Open (start closing sequence)
        IF NOT fbProcessValves2Open AND lastProcessCommand THEN
            // Start closing sequence
            isOpeningMode := FALSE;
            currentValveIndex := 1;
            numValvesInSequence := fbNumValvesToClose;
            fbSequenceActive := TRUE;
            fbSequenceComplete := FALSE;
            sequenceState := 1;  // Go to command first valve
        END_IF

        // Update edge detection variable
        lastProcessCommand := fbProcessValves2Open;


    //---------- State 1: Command Current Valve ----------//
    1:
        fbCurrentValveNum := currentValveIndex;

        // Check if we've positioned all requested valves
        IF currentValveIndex > numValvesInSequence THEN
            fbSequenceComplete := TRUE;
            sequenceState := 0;  // Return to idle
        ELSE
            // Find the valve in fbValves array
            // Use appropriate index array based on mode
            valveFound := FALSE;
            FOR i := 1 TO GVL.valveCount DO
                // Get the valve ID from the appropriate sequence array
                IF isOpeningMode THEN
                    IF fbValves[i].ID = fbValveIndexOpen[currentValveIndex] THEN
                        // Found the valve - command it to open
                        currentValveArrayPos := i;
                        fbValves[i].state := 1;
                        fbValves[i].isOpen := TRUE;
                        valveFound := TRUE;
                    END_IF
                ELSE
                    IF fbValves[i].ID = fbValveIndexClose[currentValveIndex] THEN
                        // Found the valve - command it to close
                        currentValveArrayPos := i;
                        fbValves[i].state := 1;
                        fbValves[i].isOpen := FALSE;
                        valveFound := TRUE;
                    END_IF
                END_IF

                IF valveFound THEN
                    // Capture current DI2 state for edge detection
                    lastDI2State := fbValves[i].DI2;
                    valveStartedMoving := FALSE;

                    // Reset timeout timer
                    timeoutTimer(IN := FALSE);

                    sequenceState := 2;  // Go wait for valve to start moving
                    EXIT;
                END_IF
            END_FOR

            // If valve not found in array, skip to next
            IF NOT valveFound THEN
                currentValveIndex := currentValveIndex + 1;
                // Stay in state 1 to try next valve
            END_IF
        END_IF


    //---------- State 2: Wait for Valve to Start Moving (Edge Detection) ----------//
    2:
        // DI2 is TRUE when valve is closed, FALSE when opening/open
        // Opening: Detect falling edge (TRUE -> FALSE) = valve leaving closed position
        // Closing: Detect rising edge (FALSE -> TRUE) = valve arriving at closed position

        IF isOpeningMode THEN
            // Opening mode: Wait for DI2 falling edge
            IF lastDI2State AND NOT fbValves[currentValveArrayPos].DI2 THEN
                // Falling edge detected - valve started opening
                valveStartedMoving := TRUE;
                timeoutTimer(IN := FALSE);  // Reset timeout
                delayTimer(IN := FALSE);    // Reset delay timer
                sequenceState := 3;         // Go to delay state
            END_IF
        ELSE
            // Closing mode: Wait for DI2 rising edge
            IF NOT lastDI2State AND fbValves[currentValveArrayPos].DI2 THEN
                // Rising edge detected - valve started closing (arrived at closed)
                valveStartedMoving := TRUE;
                timeoutTimer(IN := FALSE);  // Reset timeout
                delayTimer(IN := FALSE);    // Reset delay timer
                sequenceState := 3;         // Go to delay state
            END_IF
        END_IF

        // Update for next scan edge detection
        lastDI2State := fbValves[currentValveArrayPos].DI2;

        // Run timeout timer
        timeoutTimer(IN := TRUE, PT := VALVE_MOVE_TIMEOUT);

        // Check for timeout
        IF timeoutTimer.Q THEN
            // Valve didn't start moving within timeout period
            fbFaultTimeout := TRUE;
            timeoutTimer(IN := FALSE);

            // Decision: Skip to next valve or halt sequence?
            // Currently: skip to next valve
            currentValveIndex := currentValveIndex + 1;
            sequenceState := 1;
        END_IF


    //---------- State 3: Delay Timer after movement started ----------//
    3:
        // Run delay timer
        delayTimer(IN := TRUE, PT := VALVE_MOVE_DELAY);

        IF delayTimer.Q THEN
            // Delay complete
            delayTimer(IN := FALSE);  // Reset timer
            sequenceState := 4;       // Advance to next valve
        END_IF


    //---------- State 4: Advance to Next Valve ----------//
    4:
        currentValveIndex := currentValveIndex + 1;
        sequenceState := 1;  // Go back to command state for next valve


    //---------- Default: Safety ----------//
    ELSE
        sequenceState := 0;  // Return to idle if invalid state

END_CASE

END_FUNCTION_BLOCK

// ---- POUs/UnitOp FBs/FBUO_OverPressure_EX.TcPOU
FUNCTION_BLOCK FBUO_OverPressure_EX
VAR_INPUT
    fbOPprocessState 		: BOOL;
    fbValvePositionReady 	: BOOL;
	fbPumpActive 			: BOOL;
	fbPumpSpeed				: REAL;
END_VAR
VAR_IN_OUT
    fbValves : ARRAY[1..GVL.valveCount] OF ST_Valves;
END_VAR
VAR_OUTPUT
	
END_VAR
VAR
    valveIndexOpen : ARRAY[1..GVL.valveCount] OF INT := [2,4,7,8,9,10];
	numValvesToOpen : INT := 10;
	valveIndexClose : ARRAY[1..GVL.valveCount] OF INT := [2,4,7,8,9,10];
	numValvesToClose : INT := 10;
    targetState : INT;
    targetOpenClose : BOOL;
	fbValvePos : FB_ValvePOS;
	valveCtrl : FB_valveCTRL;
	valveIndex: INT;
END_VAR

IF fbOPprocessState THEN
	
	fbValvePos(fbValveIndexOpen := valveIndexOpen,
            fbNumValvesToOpen := numValvesToOpen,
			fbValveIndexClose := valveIndexClose,
            fbNumValvesToClose := numValvesToClose,
            fbValves := fbValves,
			fbProcessValves2Open := fbValvePositionReady);
    
    ValveCtrl(fbValves := fbValves);
    IO.AO1_dilutionSV := fbValves[1].AO1;
    IO.AO1_wfiSV := fbValves[2].AO1;
    IO.AO1_formDrain := fbValves[3].AO1;
    IO.AO1_wfiBypassIn := fbValves[4].AO1;
	IO.AO1_wfiFilterIn := fbValves[5].AO1;
	IO.AO1_wfiFilterOut := fbValves[6].AO1;
	IO.AO1_wfiBypassOut := fbValves[7].AO1;
	IO.AO1_dilutionDiV := fbValves[8].AO1;
	IO.AO1_FormManifold := fbValves[9].AO1;
	IO.AO1_SuspManifold := fbValves[10].AO1;
	
	
	
//-----------------------PUMP Control ----------------------//	
// 	IF fbPumpActive THEN
// 	outputAO3 := IO.AO3 := 5;
// 		GVL.DO_wfiPump := fbPumpActive;
// 		GVL.AO_wfiPump := fbPumpSpeed;
// 	ELSE
// 		GVL.DO_wfiPump := fbPumpActive;
// 		GVL.AO_wfiPump := 0;
// 	END_IF	
//---------------------------------------------------------//	
END_IF

END_FUNCTION_BLOCK

// ---- POUs/General FBs/FB_PressureMonitor.TcPOU
FUNCTION_BLOCK FB_PressureMonitor
VAR_IN_OUT
	fbSensors : ARRAY[1..GVL.pressureSensorCount] OF ST_PressureSensor;
END_VAR

VAR
	fbScale : ARRAY[1..GVL.pressureSensorCount] OF FB_ScaleAnalog;
	fbFilter : ARRAY[1..GVL.pressureSensorCount] OF FB_FirstOrderLP;
	i : INT;
END_VAR

FOR i := 1 TO GVL.pressureSensorCount DO
	// Scale raw input to engineering units
	fbScale[i](
		fbRawValue := fbSensors[i].RawValue,
		fbInputMin := fbSensors[i].InputMin,
		fbInputMax := fbSensors[i].InputMax,
		fbOutputMin := fbSensors[i].OutputMin,
		fbOutputMax := fbSensors[i].OutputMax,
		fbScaledValue => fbSensors[i].ScaledValue,
		fbRangeError => fbSensors[i].RangeError);

	// Apply low-pass filter to scaled value
	fbFilter[i](
		fbInput := fbSensors[i].ScaledValue,
		fbTimeConst := fbSensors[i].FilterTimeConst,
		fbOutput => fbSensors[i].FilteredValue);
END_FOR

END_FUNCTION_BLOCK

// ---- POUs/General FBs/FB_ScaleAnalog.TcPOU
FUNCTION_BLOCK FB_ScaleAnalog
VAR_INPUT
    fbRawValue : REAL;              // Raw analog input value (e.g., 4.0 to 20.0 mA)
    fbInputMin : REAL;              // Minimum raw input value (e.g., 4.0 for 4mA)
    fbInputMax : REAL;              // Maximum raw input value (e.g., 20.0 for 20mA)
    fbOutputMin : REAL;             // Minimum engineering unit value (e.g., 0.0 PSI)
    fbOutputMax : REAL;             // Maximum engineering unit value (e.g., 30.0 PSI)
    fbEnableLimit : BOOL := TRUE;   // Enable output limiting to min/max range
END_VAR

VAR_OUTPUT
    fbScaledValue : REAL;           // Scaled output in engineering units
    fbRangeError : BOOL;            // TRUE if input is outside expected range
    fbLimitActive : BOOL;           // TRUE if output is being limited
END_VAR

VAR
    inputRange : REAL;              // Calculated input range
    outputRange : REAL;             // Calculated output range
    normalizedValue : REAL;         // Normalized input (0.0 to 1.0)
    rawOutput : REAL;               // Output before limiting
END_VAR

// Generic Linear Scaling Function Block
// Converts raw analog input (e.g., 4-20mA) to engineering units
// Formula: Output = ((Input - InputMin) / (InputMax - InputMin)) * (OutputMax - OutputMin) + OutputMin

// Reset outputs
fbRangeError := FALSE;
fbLimitActive := FALSE;

// Calculate input and output ranges
inputRange := fbInputMax - fbInputMin;
outputRange := fbOutputMax - fbOutputMin;

// Check for invalid input range (divide by zero protection)
IF ABS(inputRange) < 0.001 THEN
    // Invalid range - return minimum output and set error
    fbScaledValue := fbOutputMin;
    fbRangeError := TRUE;
    RETURN;
END_IF

// Check if input is outside expected range
IF fbRawValue < fbInputMin OR fbRawValue > fbInputMax THEN
    fbRangeError := TRUE;
END_IF

// Normalize input to 0.0 to 1.0 range
normalizedValue := (fbRawValue - fbInputMin) / inputRange;

// Scale to output range
rawOutput := (normalizedValue * outputRange) + fbOutputMin;

// Apply limits if enabled
IF fbEnableLimit THEN
    IF rawOutput < fbOutputMin THEN
        fbScaledValue := fbOutputMin;
        fbLimitActive := TRUE;
    ELSIF rawOutput > fbOutputMax THEN
        fbScaledValue := fbOutputMax;
        fbLimitActive := TRUE;
    ELSE
        fbScaledValue := rawOutput;
    END_IF
ELSE
    // No limiting - allow values outside range
    fbScaledValue := rawOutput;
END_IF

END_FUNCTION_BLOCK

// ---- POUs/General FBs/FB_FirstOrderLP.TcPOU
FUNCTION_BLOCK FB_FirstOrderLP
VAR_INPUT
	fbInput : REAL;					// Raw input value
	fbTimeConst : REAL;				// Filter time constant in seconds (e.g., 0.1 = 100ms)
	fbCycleTime : REAL := 0.01;		// Task cycle time in seconds (default 10ms)
END_VAR

VAR_OUTPUT
	fbOutput : REAL;				// Filtered output value
END_VAR

VAR
	alpha : REAL;					// Computed filter coefficient
	bInitialized : BOOL;			// First-call flag
END_VAR

// First-Order Low-Pass Filter (Exponential Moving Average)
// Transfer: Output[n] = Output[n-1] + Alpha * (Input[n] - Output[n-1])
// Alpha = CycleTime / (TimeConst + CycleTime)

// Initialize output to first input value to avoid startup transient
IF NOT bInitialized THEN
	fbOutput := fbInput;
	bInitialized := TRUE;
	RETURN;
END_IF

// Bypass filter if time constant is zero or negative
IF fbTimeConst <= 0.0 THEN
	fbOutput := fbInput;
	RETURN;
END_IF

// Compute alpha and apply filter
alpha := fbCycleTime / (fbTimeConst + fbCycleTime);
fbOutput := fbOutput + alpha * (fbInput - fbOutput);

END_FUNCTION_BLOCK

// ---- POUs/General FBs/FB_MassFlowMonitor.TcPOU
FUNCTION_BLOCK FB_MassFlowMonitor
VAR_IN_OUT
	fbSensors : ARRAY[1..GVL.massFlowSensorCount] OF ST_MassFlowSensor;
END_VAR

VAR
	fbScale : ARRAY[1..GVL.massFlowSensorCount] OF FB_ScaleAnalog;
	i : INT;
END_VAR

FOR i := 1 TO GVL.massFlowSensorCount DO
	fbScale[i](
		fbRawValue := fbSensors[i].RawValue,
		fbInputMin := fbSensors[i].InputMin,
		fbInputMax := fbSensors[i].InputMax,
		fbOutputMin := fbSensors[i].OutputMin,
		fbOutputMax := fbSensors[i].OutputMax,
		fbScaledValue => fbSensors[i].ScaledValue,
		fbRangeError => fbSensors[i].RangeError);
END_FOR

END_FUNCTION_BLOCK

// ---- POUs/General FBs/FB_FlowPathCheck.TcPOU
FUNCTION_BLOCK FB_FlowPathCheck
VAR_IN_OUT
	fbRequiredValves : ARRAY[1..GVL.valveCount] OF INT;	// Valve indices that must be open (0 = unused slot)
	fbValves : ARRAY[1..GVL.valveCount] OF ST_Valves;		// Valve data array
END_VAR

VAR_OUTPUT
	fbPathOpen : BOOL;		// TRUE if all required valves confirmed open (DI1 = TRUE)
	fbValveCount : INT;		// Number of valves checked (non-zero entries)
END_VAR

VAR
	i : INT;
	nChecked : INT;
	bAllOpen : BOOL;
END_VAR

// Check if all required valves in the flow path are confirmed open
// A valve is confirmed open when DI1 = TRUE (open feedback)
// DI2 = TRUE means valve is closed
// Index entries of 0 are skipped (unused slots in the array)

bAllOpen := TRUE;
nChecked := 0;

FOR i := 1 TO GVL.valveCount DO
	IF fbRequiredValves[i] > 0 AND fbRequiredValves[i] <= GVL.valveCount THEN
		nChecked := nChecked + 1;
		IF NOT fbValves[fbRequiredValves[i]].DI1 THEN
			bAllOpen := FALSE;
		END_IF
	END_IF
END_FOR

// Path is only open if at least one valve was checked and all are confirmed open
fbPathOpen := bAllOpen AND (nChecked > 0);
fbValveCount := nChecked;

END_FUNCTION_BLOCK

// ---- POUs/General FBs/FB_MovingAverage.TcPOU
FUNCTION_BLOCK FB_MovingAverage
VAR_INPUT
    fbInputValue : REAL;                // Current input value to be averaged
    fbSampleSize : INT :=10;           // Number of samples in moving average (1 to 100)
    fbReset : BOOL := FALSE;            // Reset the buffer and restart averaging
END_VAR

VAR_OUTPUT
    fbAverageValue : REAL;              // Calculated moving average
    fbBufferFull : BOOL;                // TRUE when buffer has fbSampleSize valid samples
    fbValidSamples : INT;               // Current number of valid samples in buffer
END_VAR

VAR
    buffer : ARRAY[1..100] OF REAL;     // Circular buffer for samples
    bufferIndex : INT := 1;             // Current position in buffer (1 to fbSampleSize)
    sum : REAL := 0.0;                  // Running sum of all samples in buffer
    initialized : BOOL := FALSE;        // Flag for first-time initialization
    lastSampleSize : INT := 0;          // Previous sample size for change detection
    lastResetState : BOOL := FALSE;     // Previous reset state for edge detection
    i : INT;                            // Loop counter
END_VAR

// Moving Average Function Block
// Calculates running average using circular buffer
// Efficient: Only updates sum by removing old value and adding new value

// Handle reset request (rising edge detection)
IF fbReset AND NOT lastResetState THEN
    // Rising edge detected - perform reset
    FOR i := 1 TO 100 DO
        buffer[i] := 0.0;
    END_FOR
    sum := 0.0;
    bufferIndex := 1;
    fbValidSamples := 0;
    fbBufferFull := FALSE;
    initialized := FALSE;
    lastSampleSize := 0;
    fbAverageValue := 0.0;
END_IF

// Update edge detection
lastResetState := fbReset;

// If reset was just triggered, skip this scan
IF NOT initialized AND fbReset THEN
    RETURN;
END_IF

// Validate and limit sample size
IF fbSampleSize < 1 THEN
    fbSampleSize := 1;
ELSIF fbSampleSize > 100 THEN
    fbSampleSize := 100;
END_IF

// Detect sample size change and reinitialize if needed
IF fbSampleSize <> lastSampleSize AND initialized THEN
    // Sample size changed - reset and restart
    FOR i := 1 TO 100 DO
        buffer[i] := 0.0;
    END_FOR
    sum := 0.0;
    bufferIndex := 1;
    fbValidSamples := 0;
    fbBufferFull := FALSE;
    initialized := FALSE;
END_IF

lastSampleSize := fbSampleSize;

// First-time initialization
IF NOT initialized THEN
    // Fill buffer with first input value for smooth startup
    FOR i := 1 TO fbSampleSize DO
        buffer[i] := fbInputValue;
    END_FOR
    sum := fbInputValue * fbSampleSize;
    bufferIndex := 1;
    fbValidSamples := fbSampleSize;
    fbBufferFull := TRUE;
    fbAverageValue := fbInputValue;
    initialized := TRUE;
    RETURN;
END_IF

// Update moving average using circular buffer
// Remove old value from sum
sum := sum - buffer[bufferIndex];

// Add new value to buffer and sum
buffer[bufferIndex] := fbInputValue;
sum := sum + fbInputValue;

// Increment buffer index (circular)
bufferIndex := bufferIndex + 1;
IF bufferIndex > fbSampleSize THEN
    bufferIndex := 1;
    fbBufferFull := TRUE;
END_IF

// Track valid samples (during initial fill)
IF NOT fbBufferFull THEN
    fbValidSamples := bufferIndex - 1;
    IF fbValidSamples < 1 THEN
        fbValidSamples := 1;
    END_IF
ELSE
    fbValidSamples := fbSampleSize;
END_IF

// Calculate average
IF fbValidSamples > 0 THEN
    fbAverageValue := sum / fbValidSamples;
ELSE
    fbAverageValue := fbInputValue;
END_IF

END_FUNCTION_BLOCK

// ---- POUs/UnitOp FBs/FBUO_OPPump_SyringeSetup.TcPOU
FUNCTION_BLOCK FBUO_OPPump_SyringeSetup
VAR_INPUT
    bEnable         : BOOL;     // Enable the function block
    bStart          : BOOL;     // Start the setup process (rising edge)
END_VAR

VAR_OUTPUT
    bBusy           : BOOL;     // Setup in progress
    bDone           : BOOL;     // Setup complete - syringes at midpoint
    bError          : BOOL;     // Error occurred
    nCurrentStep    : INT;      // Current step for diagnostics
END_VAR

VAR
    // State machine
    nState          : INT := 0;

    // Edge detection
    rtrigStart      : R_TRIG;

    // Timing
    tonDelay        : TON;
    tonTimeout      : TON;       // Timeout for command acknowledgment

    // Tracking which axes have been stopped
    bAxis0Stopped   : BOOL;
    bAxis1Stopped   : BOOL;

    // Target volume for midpoint (ul)
    rTargetVolume   : LREAL := 12500.0;

    // Tracking fill started (saw BUSY state)
    bAxis0FillStarted : BOOL;
    bAxis1FillStarted : BOOL;

    // Tracking fill complete (saw IDLE after BUSY)
    bAxis0FillDone  : BOOL;
    bAxis1FillDone  : BOOL;

    // Tracking empty started (saw BUSY state)
    bAxis0EmptyStarted : BOOL;
    bAxis1EmptyStarted : BOOL;
END_VAR

(* FBUO_OPPump_SyringeSetup
   Purpose: Prepare syringes for operator attachment
   Process:
   1. Fill both axes until they bottom out (hit limit switch, status goes IDLE)
   2. Empty both axes until VolumeRemainingCorrected reaches 12500ul (midpoint)
   3. Stop at midpoint for operator to attach syringes

   Commands are offset by 100ms to avoid serial bus contention
   Each command waits for acknowledgment (eSelectedAction returns to IDLE) before proceeding
   Fill/Empty waits for BUSY state before waiting for IDLE (confirms motion started)
*)

// Edge detection on Start
rtrigStart(CLK := bStart AND bEnable);

// Reset outputs when disabled
IF NOT bEnable THEN
    nState := 0;
    bBusy := FALSE;
    bDone := FALSE;
    bError := FALSE;
    bAxis0Stopped := FALSE;
    bAxis1Stopped := FALSE;
    bAxis0FillStarted := FALSE;
    bAxis1FillStarted := FALSE;
    bAxis0FillDone := FALSE;
    bAxis1FillDone := FALSE;
    bAxis0EmptyStarted := FALSE;
    bAxis1EmptyStarted := FALSE;
    tonDelay(IN := FALSE);
    tonTimeout(IN := FALSE);
    RETURN;
END_IF

// State machine
CASE nState OF

    0: // IDLE - Wait for start
        nCurrentStep := 0;
        bBusy := FALSE;
        bDone := FALSE;
        bError := FALSE;
        bAxis0Stopped := FALSE;
        bAxis1Stopped := FALSE;
        bAxis0FillStarted := FALSE;
        bAxis1FillStarted := FALSE;
        bAxis0FillDone := FALSE;
        bAxis1FillDone := FALSE;
        bAxis0EmptyStarted := FALSE;
        bAxis1EmptyStarted := FALSE;

        IF rtrigStart.Q THEN
            bBusy := TRUE;
            nState := 10;
        END_IF

    // ===== FILL PHASE =====

    10: // FILL_LEFT - Send Fill command for axis 0
        nCurrentStep := 1;
        GVL_Serial.eSelectedAction := EN_AtlasPumpAction.FILL_LEFT_FAST;
        nState := 15;

    15: // WAIT_FILL_LEFT_ACK - Wait for command to be processed
        // Command is processed when eSelectedAction returns to IDLE
        IF GVL_Serial.eSelectedAction = EN_AtlasPumpAction.IDLE THEN
            tonDelay(IN := FALSE);
            nState := 20;
        END_IF

    20: // FILL_DELAY - Wait 100ms before sending next command
        tonDelay(IN := TRUE, PT := T#100MS);
        IF tonDelay.Q THEN
            tonDelay(IN := FALSE);
            nState := 30;
        END_IF

    30: // FILL_RIGHT - Send Fill command for axis 1
        nCurrentStep := 2;
        GVL_Serial.eSelectedAction := EN_AtlasPumpAction.FILL_RIGHT_FAST;
        nState := 35;

    35: // WAIT_FILL_RIGHT_ACK - Wait for command to be processed
        IF GVL_Serial.eSelectedAction = EN_AtlasPumpAction.IDLE THEN
            nState := 40;
        END_IF

    40: // WAIT_FILL_BUSY - Wait for both axes to show BUSY (confirms fill started)
        nCurrentStep := 3;

        // Check if axis 0 has started (BUSY)
        IF GVL_Serial.stPumpStatus[0].Valid AND GVL_Serial.stPumpStatus[0].IsBusy THEN
            bAxis0FillStarted := TRUE;
        END_IF

        // Check if axis 1 has started (BUSY)
        IF GVL_Serial.stPumpStatus[1].Valid AND GVL_Serial.stPumpStatus[1].IsBusy THEN
            bAxis1FillStarted := TRUE;
        END_IF

        // Both started - now wait for them to finish
        IF bAxis0FillStarted AND bAxis1FillStarted THEN
            nState := 45;
        END_IF

    45: // WAIT_FILL_IDLE - Wait for both axes to go IDLE (bottomed out)
        nCurrentStep := 4;

        // Check if axis 0 has gone IDLE (bottomed out)
        IF GVL_Serial.stPumpStatus[0].Valid AND GVL_Serial.stPumpStatus[0].IsIdle THEN
            bAxis0FillDone := TRUE;
        END_IF

        // Check if axis 1 has gone IDLE (bottomed out)
        IF GVL_Serial.stPumpStatus[1].Valid AND GVL_Serial.stPumpStatus[1].IsIdle THEN
            bAxis1FillDone := TRUE;
        END_IF

        // Both bottomed out - proceed to empty phase
        IF bAxis0FillDone AND bAxis1FillDone THEN
            tonDelay(IN := FALSE);
            nState := 50;
        END_IF

    // ===== EMPTY PHASE =====

    50: // EMPTY_LEFT - Send Empty command for axis 0
        nCurrentStep := 5;
        GVL_Serial.eSelectedAction := EN_AtlasPumpAction.EMPTY_LEFT_FAST;
        nState := 55;

    55: // WAIT_EMPTY_LEFT_ACK - Wait for command to be processed
        IF GVL_Serial.eSelectedAction = EN_AtlasPumpAction.IDLE THEN
            tonDelay(IN := FALSE);
            nState := 60;
        END_IF

    60: // EMPTY_DELAY - Wait 100ms before sending next command
        tonDelay(IN := TRUE, PT := T#100MS);
        IF tonDelay.Q THEN
            tonDelay(IN := FALSE);
            nState := 70;
        END_IF

    70: // EMPTY_RIGHT - Send Empty command for axis 1
        nCurrentStep := 6;
        GVL_Serial.eSelectedAction := EN_AtlasPumpAction.EMPTY_RIGHT_FAST;
        nState := 75;

    75: // WAIT_EMPTY_RIGHT_ACK - Wait for command to be processed
        IF GVL_Serial.eSelectedAction = EN_AtlasPumpAction.IDLE THEN
            bAxis0Stopped := FALSE;
            bAxis1Stopped := FALSE;
            nState := 76;
        END_IF

    76: // WAIT_EMPTY_BUSY - Wait for both axes to show BUSY (confirms empty started)
        nCurrentStep := 7;

        // Check if axis 0 has started (BUSY)
        IF GVL_Serial.stPumpStatus[0].Valid AND GVL_Serial.stPumpStatus[0].IsBusy THEN
            bAxis0EmptyStarted := TRUE;
        END_IF

        // Check if axis 1 has started (BUSY)
        IF GVL_Serial.stPumpStatus[1].Valid AND GVL_Serial.stPumpStatus[1].IsBusy THEN
            bAxis1EmptyStarted := TRUE;
        END_IF

        // Both started - now monitor for target volume
        IF bAxis0EmptyStarted AND bAxis1EmptyStarted THEN
            nState := 80;
        END_IF

    80: // MONITOR_EMPTY - Monitor volumes, stop whichever axis reaches midpoint first
        nCurrentStep := 8;

        // Check axis 0 - stop when VolumeRemainingCorrected <= target
        IF NOT bAxis0Stopped AND NOT bAxis1Stopped THEN
            // Neither stopped yet - check axis 0 first
            IF GVL_Serial.stPumpStatus[0].Valid AND
               GVL_Serial.stPumpStatus[0].VolumeRemainingCorrected <= rTargetVolume THEN
                GVL_Serial.eSelectedAction := EN_AtlasPumpAction.STOP_LEFT;
                bAxis0Stopped := TRUE;
                nState := 82;  // Wait for ack, then check axis 1
            // Also check axis 1 - it might reach target first
            ELSIF GVL_Serial.stPumpStatus[1].Valid AND
                  GVL_Serial.stPumpStatus[1].VolumeRemainingCorrected <= rTargetVolume THEN
                GVL_Serial.eSelectedAction := EN_AtlasPumpAction.STOP_RIGHT;
                bAxis1Stopped := TRUE;
                nState := 92;  // Wait for ack, then check axis 0
            END_IF
        ELSIF bAxis0Stopped AND NOT bAxis1Stopped THEN
            // Axis 0 already stopped, check axis 1
            IF GVL_Serial.stPumpStatus[1].Valid AND
               GVL_Serial.stPumpStatus[1].VolumeRemainingCorrected <= rTargetVolume THEN
                GVL_Serial.eSelectedAction := EN_AtlasPumpAction.STOP_RIGHT;
                bAxis1Stopped := TRUE;
                nState := 94;  // Wait for ack then done
            END_IF
        ELSIF bAxis1Stopped AND NOT bAxis0Stopped THEN
            // Axis 1 already stopped, check axis 0
            IF GVL_Serial.stPumpStatus[0].Valid AND
               GVL_Serial.stPumpStatus[0].VolumeRemainingCorrected <= rTargetVolume THEN
                GVL_Serial.eSelectedAction := EN_AtlasPumpAction.STOP_LEFT;
                bAxis0Stopped := TRUE;
                nState := 94;  // Wait for ack then done
            END_IF
        END_IF

        // Both stopped - done
        IF bAxis0Stopped AND bAxis1Stopped THEN
            nState := 100;
        END_IF

    82: // WAIT_STOP_LEFT_ACK - Wait for stop command to be processed
        IF GVL_Serial.eSelectedAction = EN_AtlasPumpAction.IDLE THEN
            tonDelay(IN := FALSE);
            nState := 85;
        END_IF

    85: // STOP_DELAY_0 - Wait 100ms after stopping axis 0
        tonDelay(IN := TRUE, PT := T#100MS);
        IF tonDelay.Q THEN
            tonDelay(IN := FALSE);
            // Go back to monitor to check axis 1
            nState := 80;
        END_IF

    92: // WAIT_STOP_RIGHT_ACK - Wait for stop command to be processed
        IF GVL_Serial.eSelectedAction = EN_AtlasPumpAction.IDLE THEN
            tonDelay(IN := FALSE);
            nState := 93;
        END_IF

    93: // STOP_DELAY_1 - Wait 100ms after stopping axis 1
        tonDelay(IN := TRUE, PT := T#100MS);
        IF tonDelay.Q THEN
            tonDelay(IN := FALSE);
            // Go back to monitor to check axis 0
            nState := 80;
        END_IF

    94: // WAIT_FINAL_STOP_ACK - Wait for final stop command to be processed
        nCurrentStep := 9;
        IF GVL_Serial.eSelectedAction = EN_AtlasPumpAction.IDLE THEN
            nState := 100;
        END_IF

    // ===== COMPLETE =====

    100: // DONE - Setup complete
        nCurrentStep := 10;
        bBusy := FALSE;
        bDone := TRUE;

        // Wait for bStart to go FALSE before allowing restart
        IF NOT bStart THEN
            nState := 0;
        END_IF

END_CASE

END_FUNCTION_BLOCK

// ---- POUs/UnitOp FBs/FBUO_OPPUMP_AcetonePrime.TcPOU
FUNCTION_BLOCK FBUO_OPPump_AcetonePrime
VAR_INPUT
    bEnable             : BOOL;         // Enable the function block
    bStartAcetonePrime  : BOOL;         // Start the priming process (rising edge)
    nSyringeCycles      : INT := 2;     // Number of fill/empty cycles
END_VAR

VAR_OUTPUT
    bBusy               : BOOL;         // Priming in progress
    bDone               : BOOL;         // Priming complete
    bError              : BOOL;         // Error occurred
    nCurrentStep        : INT;          // Current step for diagnostics
    nCurrentCycle       : INT;          // Current cycle number (1 to nSyringeCycles)
END_VAR

VAR
    // State machine
    nState              : INT := 0;

    // Edge detection
    rtrigStart          : R_TRIG;

    // Timing
    tonDelay            : TON;

    // Cycle counter
    nCycleCount         : INT := 0;

    // Tracking fill started (saw BUSY state)
    bAxis0FillStarted   : BOOL;
    bAxis1FillStarted   : BOOL;

    // Tracking fill complete (saw IDLE after BUSY)
    bAxis0FillDone      : BOOL;
    bAxis1FillDone      : BOOL;

    // Tracking empty started (saw BUSY state)
    bAxis0EmptyStarted  : BOOL;
    bAxis1EmptyStarted  : BOOL;

    // Tracking empty complete (saw IDLE after BUSY)
    bAxis0EmptyDone     : BOOL;
    bAxis1EmptyDone     : BOOL;
END_VAR

(* FBUO_OPPump_AcetonePrime
   Purpose: Prime syringes with acetone (or other solvent)
   Process:
   1. Fill both syringes (wait for IDLE)
   2. Empty both syringes (wait for IDLE)
   3. Repeat for nSyringeCycles times
   4. End with syringes empty after last cycle

   Commands are offset by 100ms to avoid serial bus contention
   Uses _PRIME speed commands
*)

// Edge detection on Start
rtrigStart(CLK := bStartAcetonePrime AND bEnable);

// Reset outputs when disabled
IF NOT bEnable THEN
    nState := 0;
    bBusy := FALSE;
    bDone := FALSE;
    bError := FALSE;
    nCycleCount := 0;
    nCurrentCycle := 0;
    bAxis0FillStarted := FALSE;
    bAxis1FillStarted := FALSE;
    bAxis0FillDone := FALSE;
    bAxis1FillDone := FALSE;
    bAxis0EmptyStarted := FALSE;
    bAxis1EmptyStarted := FALSE;
    bAxis0EmptyDone := FALSE;
    bAxis1EmptyDone := FALSE;
    tonDelay(IN := FALSE);
    RETURN;
END_IF

// State machine
CASE nState OF

    0: // IDLE - Wait for start
        nCurrentStep := 0;
        nCurrentCycle := 0;
        bBusy := FALSE;
        bDone := FALSE;
        bError := FALSE;
        nCycleCount := 0;

        IF rtrigStart.Q THEN
            bBusy := TRUE;
            nCycleCount := 1;
            nCurrentCycle := 1;
            nState := 10;
        END_IF

    // ===== FILL PHASE =====

    10: // FILL_LEFT - Send Fill command for axis 0
        nCurrentStep := 1;
        // Reset tracking flags for this cycle
        bAxis0FillStarted := FALSE;
        bAxis1FillStarted := FALSE;
        bAxis0FillDone := FALSE;
        bAxis1FillDone := FALSE;
        GVL_Serial.eSelectedAction := EN_AtlasPumpAction.FILL_LEFT_PRIME;
        nState := 15;

    15: // WAIT_FILL_LEFT_ACK - Wait for command to be processed
        IF GVL_Serial.eSelectedAction = EN_AtlasPumpAction.IDLE THEN
            tonDelay(IN := FALSE);
            nState := 20;
        END_IF

    20: // FILL_DELAY - Wait 100ms before sending next command
        tonDelay(IN := TRUE, PT := T#100MS);
        IF tonDelay.Q THEN
            tonDelay(IN := FALSE);
            nState := 30;
        END_IF

    30: // FILL_RIGHT - Send Fill command for axis 1
        nCurrentStep := 2;
        GVL_Serial.eSelectedAction := EN_AtlasPumpAction.FILL_RIGHT_PRIME;
        nState := 35;

    35: // WAIT_FILL_RIGHT_ACK - Wait for command to be processed
        IF GVL_Serial.eSelectedAction = EN_AtlasPumpAction.IDLE THEN
            nState := 40;
        END_IF

    40: // WAIT_FILL_BUSY - Wait for both axes to show BUSY (confirms fill started)
        nCurrentStep := 3;

        // Check if axis 0 has started (BUSY)
        IF GVL_Serial.stPumpStatus[0].Valid AND GVL_Serial.stPumpStatus[0].IsBusy THEN
            bAxis0FillStarted := TRUE;
        END_IF

        // Check if axis 1 has started (BUSY)
        IF GVL_Serial.stPumpStatus[1].Valid AND GVL_Serial.stPumpStatus[1].IsBusy THEN
            bAxis1FillStarted := TRUE;
        END_IF

        // Both started - now wait for them to finish
        IF bAxis0FillStarted AND bAxis1FillStarted THEN
            nState := 45;
        END_IF

    45: // WAIT_FILL_IDLE - Wait for both axes to go IDLE (fill complete)
        nCurrentStep := 4;

        // Check if axis 0 has gone IDLE (fill complete)
        IF GVL_Serial.stPumpStatus[0].Valid AND GVL_Serial.stPumpStatus[0].IsIdle THEN
            bAxis0FillDone := TRUE;
        END_IF

        // Check if axis 1 has gone IDLE (fill complete)
        IF GVL_Serial.stPumpStatus[1].Valid AND GVL_Serial.stPumpStatus[1].IsIdle THEN
            bAxis1FillDone := TRUE;
        END_IF

        // Both fill complete - proceed to empty phase
        IF bAxis0FillDone AND bAxis1FillDone THEN
            tonDelay(IN := FALSE);
            nState := 50;
        END_IF

    // ===== EMPTY PHASE =====

    50: // EMPTY_LEFT - Send Empty command for axis 0
        nCurrentStep := 5;
        // Reset tracking flags for empty phase
        bAxis0EmptyStarted := FALSE;
        bAxis1EmptyStarted := FALSE;
        bAxis0EmptyDone := FALSE;
        bAxis1EmptyDone := FALSE;
        GVL_Serial.eSelectedAction := EN_AtlasPumpAction.EMPTY_LEFT_PRIME;
        nState := 55;

    55: // WAIT_EMPTY_LEFT_ACK - Wait for command to be processed
        IF GVL_Serial.eSelectedAction = EN_AtlasPumpAction.IDLE THEN
            tonDelay(IN := FALSE);
            nState := 60;
        END_IF

    60: // EMPTY_DELAY - Wait 100ms before sending next command
        tonDelay(IN := TRUE, PT := T#100MS);
        IF tonDelay.Q THEN
            tonDelay(IN := FALSE);
            nState := 70;
        END_IF

    70: // EMPTY_RIGHT - Send Empty command for axis 1
        nCurrentStep := 6;
        GVL_Serial.eSelectedAction := EN_AtlasPumpAction.EMPTY_RIGHT_PRIME;
        nState := 75;

    75: // WAIT_EMPTY_RIGHT_ACK - Wait for command to be processed
        IF GVL_Serial.eSelectedAction = EN_AtlasPumpAction.IDLE THEN
            nState := 76;
        END_IF

    76: // WAIT_EMPTY_BUSY - Wait for both axes to show BUSY (confirms empty started)
        nCurrentStep := 7;

        // Check if axis 0 has started (BUSY)
        IF GVL_Serial.stPumpStatus[0].Valid AND GVL_Serial.stPumpStatus[0].IsBusy THEN
            bAxis0EmptyStarted := TRUE;
        END_IF

        // Check if axis 1 has started (BUSY)
        IF GVL_Serial.stPumpStatus[1].Valid AND GVL_Serial.stPumpStatus[1].IsBusy THEN
            bAxis1EmptyStarted := TRUE;
        END_IF

        // Both started - now wait for them to finish
        IF bAxis0EmptyStarted AND bAxis1EmptyStarted THEN
            nState := 78;
        END_IF

    78: // WAIT_EMPTY_IDLE - Wait for both axes to go IDLE (empty complete)
        nCurrentStep := 8;

        // Check if axis 0 has gone IDLE (empty complete)
        IF GVL_Serial.stPumpStatus[0].Valid AND GVL_Serial.stPumpStatus[0].IsIdle THEN
            bAxis0EmptyDone := TRUE;
        END_IF

        // Check if axis 1 has gone IDLE (empty complete)
        IF GVL_Serial.stPumpStatus[1].Valid AND GVL_Serial.stPumpStatus[1].IsIdle THEN
            bAxis1EmptyDone := TRUE;
        END_IF

        // Both empty complete - check if more cycles needed
        IF bAxis0EmptyDone AND bAxis1EmptyDone THEN
            nState := 80;
        END_IF

    // ===== CYCLE CHECK =====

    80: // CHECK_CYCLES - Check if more cycles needed
        nCurrentStep := 9;

        IF nCycleCount < nSyringeCycles THEN
            // More cycles needed - increment and go back to fill
            nCycleCount := nCycleCount + 1;
            nCurrentCycle := nCycleCount;
            nState := 10;
        ELSE
            // All cycles complete - done (syringes are empty)
            nState := 100;
        END_IF

    // ===== COMPLETE =====

    100: // DONE - Priming complete
        nCurrentStep := 10;
        bBusy := FALSE;
        bDone := TRUE;

        // Wait for bStartAcetonePrime to go FALSE before allowing restart
        IF NOT bStartAcetonePrime THEN
            nState := 0;
        END_IF

END_CASE

END_FUNCTION_BLOCK

// ---- POUs/UnitOp FBs/FBUO_OPFlowFormation.TcPOU
FUNCTION_BLOCK FBUO_OPFlowFormation
VAR_INPUT
	bEnable         : BOOL;     // Enable the function block
	bStart          : BOOL;     // TRUE = run continuous flow, FALSE = stop
END_VAR

VAR_OUTPUT
	bBusy           : BOOL;     // State machine active (starting or stopping)
	bRunning        : BOOL;     // TRUE when pump is actively in continuous flow
	bError          : BOOL;     // Error occurred
	nCurrentStep    : INT;      // Current step for diagnostics
END_VAR

VAR
	nState          : INT := 0;
	rtrigStart      : R_TRIG;   // Detect rising edge of bStart
	ftrigStart      : F_TRIG;   // Detect falling edge of bStart
	tonDelay        : TON;      // Delay between stop commands
END_VAR

(* FBUO_OPFlowFormation
   Purpose: Start/stop continuous flow on the Atlas pump
   - Rising edge of bStart: sends CONTINUOUS command
   - Falling edge of bStart: sends STOP_LEFT, waits 100ms, sends STOP_RIGHT
   - The Atlas pump firmware handles all syringe alternation internally
*)

// Edge detection
rtrigStart(CLK := bStart AND bEnable);
ftrigStart(CLK := bStart AND bEnable);

// Reset when disabled
IF NOT bEnable THEN
	nState := 0;
	bBusy := FALSE;
	bRunning := FALSE;
	bError := FALSE;
	nCurrentStep := 0;
	tonDelay(IN := FALSE);
	RETURN;
END_IF

CASE nState OF

	0: // IDLE - wait for start
		nCurrentStep := 0;
		bBusy := FALSE;
		bError := FALSE;

		IF rtrigStart.Q THEN
			bBusy := TRUE;
			nState := 10;
		END_IF

	// ===== START PHASE =====

	10: // SEND_CONTINUOUS - send continuous flow command
		nCurrentStep := 1;
		GVL_Serial.eSelectedAction := EN_AtlasPumpAction.CONTINUOUS;
		nState := 15;

	15: // WAIT_ACK - wait for command to be processed by SerialComm
		IF GVL_Serial.eSelectedAction = EN_AtlasPumpAction.IDLE THEN
			bBusy := FALSE;
			bRunning := TRUE;
			nState := 20;
		END_IF

	// ===== RUNNING PHASE =====

	20: // RUNNING - pump is in continuous flow, wait for stop signal
		nCurrentStep := 2;

		IF ftrigStart.Q THEN
			bRunning := FALSE;
			bBusy := TRUE;
			nState := 30;
		END_IF

	// ===== STOP PHASE =====

	30: // STOP_LEFT - send stop command for axis 0
		nCurrentStep := 3;
		GVL_Serial.eSelectedAction := EN_AtlasPumpAction.STOP_LEFT;
		nState := 35;

	35: // WAIT_STOP_LEFT_ACK
		IF GVL_Serial.eSelectedAction = EN_AtlasPumpAction.IDLE THEN
			tonDelay(IN := FALSE);
			nState := 40;
		END_IF

	40: // STOP_DELAY - 100ms between stop commands to avoid serial contention
		tonDelay(IN := TRUE, PT := T#100MS);
		IF tonDelay.Q THEN
			tonDelay(IN := FALSE);
			nState := 50;
		END_IF

	50: // STOP_RIGHT - send stop command for axis 1
		nCurrentStep := 4;
		GVL_Serial.eSelectedAction := EN_AtlasPumpAction.STOP_RIGHT;
		nState := 55;

	55: // WAIT_STOP_RIGHT_ACK
		IF GVL_Serial.eSelectedAction = EN_AtlasPumpAction.IDLE THEN
			bBusy := FALSE;
			nState := 0;
		END_IF

END_CASE

END_FUNCTION_BLOCK

// ---- POUs/SerialComm.TcPOU
PROGRAM SerialComm
VAR
	(* background communication with the PC COM port device *)
	(* Background ADS Control *)
	fbSerialLineControlADS 	: SerialLineControlADS;
	stSerialConfig 			: ComSerialConfig; (* Using the struct above *)
	PumpCmds				: ST_AtlasPumpCmd;
	//eSelectedAction 		: EN_AtlasPumpAction := EN_AtlasPumpAction.IDLE;

	(* Status Outputs from the block *)
    bPortOpened            : BOOL;
    bError                 : BOOL;
    nErrorID               : UDINT;

	(* Command Logic *)
    fbSend            : SendString;
    fbReceive         : ReceiveString;

	(* Initialization flag *)
    bInitialized           : BOOL := FALSE;

    (* Inputs/Outputs *)
	iState            	: INT := 0;
	sCommandToSend  	: STRING;
    sResponse         	: STRING;       // Holds the received response
    bReceived         	: BOOL;         // Flashes TRUE when a message arrives
    tonTimeout        	: TON;          // To catch if the device never responds
	sCleanResponse		: STRING;

	(* PC Control Entry/Exit *)
	bInPCControl		: BOOL := FALSE;	// TRUE when pump confirmed in PC Control mode
	bIsEntryCommand		: BOOL := FALSE;	// TRUE if current command is A1 entry
	ftrigPCControl		: F_TRIG;			// Falling edge detection for bEnablePCControl
	bExitingPCControl	: BOOL := FALSE;	// TRUE while sending A0 exit command
	bIsExitCommand		: BOOL := FALSE;	// TRUE if current command is A0 exit
	sActiveCommand		: STRING;			// The command currently being sent

	(* Status Polling - replaces heartbeat once in PC Control *)
	tonStatusPoll		: TON;				// 50ms interval timer for status polling
	nStatusAxis			: INT := 0;			// Current axis to poll (alternates 0, 1)
	bIsStatusCommand	: BOOL := FALSE;	// TRUE if current command is status query

	(* Status Parsing *)
	sParseBuffer		: STRING;			// Working buffer for parsing
	nSpacePos			: INT;				// Position of space in parse buffer
	sToken				: STRING;			// Extracted token
	nFieldIndex			: INT;				// Current field being parsed
	nParsedAxis			: INT;				// Axis number parsed from response

	(* Manual Command Status *)
	bCommandDone		: BOOL := FALSE;	// Pulses TRUE when manual command completes
	bCommandTimeout		: BOOL := FALSE;	// TRUE if last manual command timed out

END_VAR

// 1. Set configuration values (Run only once)
IF NOT bInitialized THEN
    stSerialConfig.ComPort    := 8;            // Matches your USB adapter
    stSerialConfig.Baudrate   := 57600;
    stSerialConfig.Parity     := PARITY_NONE;
    stSerialConfig.DataBits   := 8;
    stSerialConfig.StopBits   := STOPBITS_ONE;

    // CRITICAL: Prevent USB blocking by enabling these
    stSerialConfig.DTR        := DTR_CTRL_ENABLE;
    stSerialConfig.RTS        := RTS_CTRL_ENABLE;

    bInitialized := TRUE;
END_IF

// Detect falling edge of bEnablePCControl to trigger A0 exit command
ftrigPCControl(CLK := GVL_Serial.bEnablePCControl);
IF ftrigPCControl.Q AND bInPCControl THEN
    bExitingPCControl := TRUE;  // Flag to send A0 command
END_IF

// Clear status polling when PC Control disabled
IF NOT GVL_Serial.bEnablePCControl AND NOT bExitingPCControl THEN
    tonStatusPoll(IN := FALSE);
    GVL_Serial.bStatusPollingActive := FALSE;
END_IF

(* 1. ALWAYS run the background communication first *)
fbSerialLineControlADS(
    Connect  := TRUE,
    SerialCfg:= stSerialConfig,
    NetId    := '',                      	(* Local CX5330 *)
    Timeout  := T#5S,
    TxBuffer := GVL_Serial.TxBufferPcCom,
    RxBuffer := GVL_Serial.RxBufferPcCom,
    PortOpened => bPortOpened,
    Error      => bError,
    ErrorID    => nErrorID);

(* 2. Status poll timer - runs when in PC Control, state machine is idle, and no manual command pending *)
tonStatusPoll(IN := bInPCControl AND bPortOpened AND (iState = 0) AND NOT GVL_Serial.bStartCommand AND GVL_Serial.eSelectedAction = EN_AtlasPumpAction.IDLE, PT := T#50MS);

(* 3. Command State Machine *)
CASE iState OF
    0: (* IDLE - Priority: Exit > Manual > Status Poll > Entry *)
        bCommandDone := FALSE;  // Clear completion flag

        // A0 Exit command takes highest priority
        IF bExitingPCControl AND bPortOpened THEN
            bIsEntryCommand  := FALSE;
            bIsExitCommand   := TRUE;
            bIsStatusCommand := FALSE;
            sActiveCommand   := 'A0$R$L';
            sResponse        := '';
            iState           := 10;

        // Manual command via enum selection
        ELSIF GVL_Serial.eSelectedAction <> EN_AtlasPumpAction.IDLE AND bPortOpened THEN
            (* Map the Selection to the specific Struct String *)
            CASE GVL_Serial.eSelectedAction OF
                EN_AtlasPumpAction.STOP_LEFT			:sCommandToSend := PumpCmds.StopLeft;
                EN_AtlasPumpAction.STOP_RIGHT			:sCommandToSend := PumpCmds.StopRight;
                EN_AtlasPumpAction.PAUSE_LEFT			:sCommandToSend := PumpCmds.PauseLeft;
                EN_AtlasPumpAction.PAUSE_RIGHT			:sCommandToSend := PumpCmds.PauseRight;
                EN_AtlasPumpAction.UNPAUSE_LEFT			:sCommandToSend := PumpCmds.UnpauseLeft;
                EN_AtlasPumpAction.UNPAUSE_RIGHT		:sCommandToSend := PumpCmds.UnpauseRight;
                EN_AtlasPumpAction.EMPTY_LEFT_FAST		:sCommandToSend := PumpCmds.EmptyLeft_FAST;
                EN_AtlasPumpAction.EMPTY_RIGHT_FAST		:sCommandToSend := PumpCmds.EmptyRight_FAST;
                EN_AtlasPumpAction.FILL_LEFT_FAST		:sCommandToSend := PumpCmds.FillLeft_FAST;
                EN_AtlasPumpAction.FILL_RIGHT_FAST		:sCommandToSend := PumpCmds.FillRight_FAST;
				EN_AtlasPumpAction.EMPTY_LEFT_PRIME		:sCommandToSend := PumpCmds.EmptyLeft_PRIME;
                EN_AtlasPumpAction.EMPTY_RIGHT_PRIME	:sCommandToSend := PumpCmds.EmptyRight_PRIME;
                EN_AtlasPumpAction.FILL_LEFT_PRIME		:sCommandToSend := PumpCmds.FillLeft_PRIME;
                EN_AtlasPumpAction.FILL_RIGHT_PRIME		:sCommandToSend := PumpCmds.FillRight_PRIME;
				EN_AtlasPumpAction.CONTINUOUS			:sCommandToSend := PumpCmds.CONTINUOUS;
            END_CASE
            GVL_Serial.eSelectedAction := EN_AtlasPumpAction.IDLE;  // Clear selection
            bIsEntryCommand  := FALSE;
            bIsExitCommand   := FALSE;
            bIsStatusCommand := FALSE;
            bCommandTimeout  := FALSE;
            sActiveCommand   := CONCAT(sCommandToSend, '$R$L');
            sResponse        := '';
            iState           := 10;

        // Manual command via bStartCommand trigger
        ELSIF GVL_Serial.bStartCommand AND bPortOpened THEN
            GVL_Serial.bStartCommand := FALSE;
            bIsEntryCommand  := FALSE;
            bIsExitCommand   := FALSE;
            bIsStatusCommand := FALSE;
            bCommandTimeout  := FALSE;
            sActiveCommand   := CONCAT(sCommandToSend, '$R$L');
            sResponse        := '';
            iState           := 10;

        // Status polling - once in PC Control, poll S0/S1 alternately every 50ms
        ELSIF bInPCControl AND bPortOpened AND tonStatusPoll.Q THEN
            tonStatusPoll(IN := FALSE);  // Reset timer
            bIsEntryCommand  := FALSE;
            bIsExitCommand   := FALSE;
            bIsStatusCommand := TRUE;
            // Alternate between S0 and S1
            IF nStatusAxis = 0 THEN
                sActiveCommand := 'S0$R$L';
            ELSE
                sActiveCommand := 'S1$R$L';
            END_IF
            sResponse := '';
            iState    := 10;
            GVL_Serial.bStatusPollingActive := TRUE;

        // A1 Entry command - only when PC Control requested but not yet confirmed
        ELSIF GVL_Serial.bEnablePCControl AND NOT bInPCControl AND bPortOpened THEN
            bIsEntryCommand  := TRUE;
            bIsExitCommand   := FALSE;
            bIsStatusCommand := FALSE;
            sActiveCommand   := 'A1$R$L';
            sResponse        := '';
            iState           := 10;
        END_IF

    10: (* SEND command *)
        fbSend(
            SendString := sActiveCommand,
            TxBuffer   := GVL_Serial.TxBufferPcCom);

        IF NOT fbSend.Busy THEN
            iState := 20;
        END_IF

    20: (* WAIT FOR RESPONSE *)
        fbReceive(
            Prefix         := '',
            Suffix         := '$R$L',
            Timeout        := T#1S,
            ReceivedString := sResponse,
            RxBuffer       := GVL_Serial.RxBufferPcCom,
            StringReceived => bReceived);

        tonTimeout(IN := TRUE, PT := T#2S);

        IF bReceived THEN
            tonTimeout(IN := FALSE);
            // Remove trailing CR/LF from response
            sCleanResponse := LEFT(sResponse, LEN(sResponse) - 2);

            // Check if this was an exit command (A0)
            IF bIsExitCommand THEN
                // A0 response is "#A" - check if we got it
                IF sCleanResponse = '#A' THEN
                    bInPCControl := FALSE;
                    GVL_Serial.bStatusPollingActive := FALSE;
                END_IF
                bExitingPCControl := FALSE;
                bIsExitCommand := FALSE;

            // Check if this was an entry command (A1)
            ELSIF bIsEntryCommand THEN
                // A1 response is "#A" - check if we got it
                IF sCleanResponse = '#A' THEN
                    bInPCControl := TRUE;
                    nStatusAxis := 0;  // Start polling with axis 0
                END_IF
                bIsEntryCommand := FALSE;

            // Check if this was a status command (S0 or S1)
            ELSIF bIsStatusCommand THEN
                // Parse the status response and populate the struct
                // Response format: #Sn <error> <state> <vol_remain> <movements> <cumul_vol> <flow_rate> <node1> <node2> <total_cumul>
                ParseStatusResponse();
                // Alternate axis for next poll
                IF nStatusAxis = 0 THEN
                    nStatusAxis := 1;
                ELSE
                    nStatusAxis := 0;
                END_IF
                bIsStatusCommand := FALSE;

            ELSE
                // Manual command completed successfully
                bCommandDone := TRUE;
            END_IF
            iState := 0;

        ELSIF tonTimeout.Q THEN
            tonTimeout(IN := FALSE);
            // Timeout handling
            IF bIsExitCommand THEN
                // Exit command timed out - clear flags anyway
                bExitingPCControl := FALSE;
                bIsExitCommand := FALSE;
                bInPCControl := FALSE;
                GVL_Serial.bStatusPollingActive := FALSE;
            ELSIF bIsEntryCommand THEN
                // Entry command timed out
                bIsEntryCommand := FALSE;
                bInPCControl := FALSE;
            ELSIF bIsStatusCommand THEN
                // Status poll timed out - mark status as invalid
                GVL_Serial.stPumpStatus[nStatusAxis].Valid := FALSE;
                // Still alternate axis
                IF nStatusAxis = 0 THEN
                    nStatusAxis := 1;
                ELSE
                    nStatusAxis := 0;
                END_IF
                bIsStatusCommand := FALSE;
            ELSE
                // Manual command timed out
                bCommandTimeout := TRUE;
                bCommandDone := TRUE;
            END_IF
            iState := 0;
        END_IF
END_CASE

ACTION ParseStatusResponse:
(* Parse status response: #Sn <error> <state> <vol_remain> <movements> <cumul_vol> <flow_rate> <node1> <node2> <total_cumul> *)
(* Example: #S0 0 6 0 0 0 0 ? ? 0 *)

// Verify response starts with "#S"
IF LEFT(sCleanResponse, 2) <> '#S' THEN
    GVL_Serial.stPumpStatus[nStatusAxis].Valid := FALSE;
    RETURN;
END_IF

// Extract axis number from position 3 (e.g., "#S0" -> "0")
nParsedAxis := STRING_TO_INT(MID(sCleanResponse, 1, 3));

// Validate axis is 0 or 1
IF nParsedAxis < 0 OR nParsedAxis > 1 THEN
    GVL_Serial.stPumpStatus[nStatusAxis].Valid := FALSE;
    RETURN;
END_IF

// Skip header "#Sn " (4 characters) to get data portion
IF LEN(sCleanResponse) <= 4 THEN
    GVL_Serial.stPumpStatus[nParsedAxis].Valid := FALSE;
    RETURN;
END_IF
sParseBuffer := RIGHT(sCleanResponse, LEN(sCleanResponse) - 4);
nFieldIndex := 0;

// Parse each space-delimited field
WHILE LEN(sParseBuffer) > 0 DO
    nSpacePos := FIND(sParseBuffer, ' ');

    IF nSpacePos > 0 THEN
        // Extract token before space
        sToken := LEFT(sParseBuffer, nSpacePos - 1);
        // Remove token and space from buffer
        sParseBuffer := RIGHT(sParseBuffer, LEN(sParseBuffer) - nSpacePos);
    ELSE
        // Last token (no more spaces)
        sToken := sParseBuffer;
        sParseBuffer := '';
    END_IF

    // Assign token to appropriate field based on index
    CASE nFieldIndex OF
        0: // Error code
            GVL_Serial.stPumpStatus[nParsedAxis].ErrorCode := STRING_TO_INT(sToken);
            GVL_Serial.stPumpStatus[nParsedAxis].HasError := (GVL_Serial.stPumpStatus[nParsedAxis].ErrorCode <> 0);

